;FOLD LIN P413 Vel=2 m/s CPDAT413 Tool[1]:marker Base[0] ;%{PE}
;FOLD Parameters ;%{h}
;Params IlfProvider=kukaroboter.basistech.inlineforms.movement.old; Kuka.IsGlobalPoint=False; Kuka.PointName=P413; Kuka.BlendingEnabled=False; Kuka.MoveDataName=CPDAT1; Kuka.VelocityPath=2; Kuka.CurrentCDSetIndex=0; Kuka.MovementParameterFieldEnabled=True; IlfCommand=LIN
;ENDFOLD
$BWDSTART = FALSE
LDAT_ACT = LCPDAT413
FDAT_ACT = FP413
BAS(#CP_PARAMS, 2.0)
SET_CD_PARAMS (0)
LIN XP413
;ENDFOLD

;FOLD LIN P414 Vel=2 m/s CPDAT414 Tool[1]:marker Base[0] ;%{PE}
;FOLD Parameters ;%{h}
;Params IlfProvider=kukaroboter.basistech.inlineforms.movement.old; Kuka.IsGlobalPoint=False; Kuka.PointName=P414; Kuka.BlendingEnabled=False; Kuka.MoveDataName=CPDAT1; Kuka.VelocityPath=2; Kuka.CurrentCDSetIndex=0; Kuka.MovementParameterFieldEnabled=True; IlfCommand=LIN
;ENDFOLD
$BWDSTART = FALSE
LDAT_ACT = LCPDAT414
FDAT_ACT = FP414
BAS(#CP_PARAMS, 2.0)
SET_CD_PARAMS (0)
LIN XP414
;ENDFOLD

;FOLD LIN P415 Vel=2 m/s CPDAT415 Tool[1]:marker Base[0] ;%{PE}
;FOLD Parameters ;%{h}
;Params IlfProvider=kukaroboter.basistech.inlineforms.movement.old; Kuka.IsGlobalPoint=False; Kuka.PointName=P415; Kuka.BlendingEnabled=False; Kuka.MoveDataName=CPDAT1; Kuka.VelocityPath=2; Kuka.CurrentCDSetIndex=0; Kuka.MovementParameterFieldEnabled=True; IlfCommand=LIN
;ENDFOLD
$BWDSTART = FALSE
LDAT_ACT = LCPDAT415
FDAT_ACT = FP415
BAS(#CP_PARAMS, 2.0)
SET_CD_PARAMS (0)
LIN XP415
;ENDFOLD

;FOLD LIN P416 Vel=2 m/s CPDAT416 Tool[1]:marker Base[0] ;%{PE}
;FOLD Parameters ;%{h}
;Params IlfProvider=kukaroboter.basistech.inlineforms.movement.old; Kuka.IsGlobalPoint=False; Kuka.PointName=P416; Kuka.BlendingEnabled=False; Kuka.MoveDataName=CPDAT1; Kuka.VelocityPath=2; Kuka.CurrentCDSetIndex=0; Kuka.MovementParameterFieldEnabled=True; IlfCommand=LIN
;ENDFOLD
$BWDSTART = FALSE
LDAT_ACT = LCPDAT416
FDAT_ACT = FP416
BAS(#CP_PARAMS, 2.0)
SET_CD_PARAMS (0)
LIN XP416
;ENDFOLD

;FOLD LIN P417 Vel=2 m/s CPDAT417 Tool[1]:marker Base[0] ;%{PE}
;FOLD Parameters ;%{h}
;Params IlfProvider=kukaroboter.basistech.inlineforms.movement.old; Kuka.IsGlobalPoint=False; Kuka.PointName=P417; Kuka.BlendingEnabled=False; Kuka.MoveDataName=CPDAT1; Kuka.VelocityPath=2; Kuka.CurrentCDSetIndex=0; Kuka.MovementParameterFieldEnabled=True; IlfCommand=LIN
;ENDFOLD
$BWDSTART = FALSE
LDAT_ACT = LCPDAT417
FDAT_ACT = FP417
BAS(#CP_PARAMS, 2.0)
SET_CD_PARAMS (0)
LIN XP417
;ENDFOLD

;FOLD LIN P418 Vel=2 m/s CPDAT418 Tool[1]:marker Base[0] ;%{PE}
;FOLD Parameters ;%{h}
;Params IlfProvider=kukaroboter.basistech.inlineforms.movement.old; Kuka.IsGlobalPoint=False; Kuka.PointName=P418; Kuka.BlendingEnabled=False; Kuka.MoveDataName=CPDAT1; Kuka.VelocityPath=2; Kuka.CurrentCDSetIndex=0; Kuka.MovementParameterFieldEnabled=True; IlfCommand=LIN
;ENDFOLD
$BWDSTART = FALSE
LDAT_ACT = LCPDAT418
FDAT_ACT = FP418
BAS(#CP_PARAMS, 2.0)
SET_CD_PARAMS (0)
LIN XP418
;ENDFOLD

;FOLD LIN P419 Vel=2 m/s CPDAT419 Tool[1]:marker Base[0] ;%{PE}
;FOLD Parameters ;%{h}
;Params IlfProvider=kukaroboter.basistech.inlineforms.movement.old; Kuka.IsGlobalPoint=False; Kuka.PointName=P419; Kuka.BlendingEnabled=False; Kuka.MoveDataName=CPDAT1; Kuka.VelocityPath=2; Kuka.CurrentCDSetIndex=0; Kuka.MovementParameterFieldEnabled=True; IlfCommand=LIN
;ENDFOLD
$BWDSTART = FALSE
LDAT_ACT = LCPDAT419
FDAT_ACT = FP419
BAS(#CP_PARAMS, 2.0)
SET_CD_PARAMS (0)
LIN XP419
;ENDFOLD

;FOLD LIN P420 Vel=2 m/s CPDAT420 Tool[1]:marker Base[0] ;%{PE}
;FOLD Parameters ;%{h}
;Params IlfProvider=kukaroboter.basistech.inlineforms.movement.old; Kuka.IsGlobalPoint=False; Kuka.PointName=P420; Kuka.BlendingEnabled=False; Kuka.MoveDataName=CPDAT1; Kuka.VelocityPath=2; Kuka.CurrentCDSetIndex=0; Kuka.MovementParameterFieldEnabled=True; IlfCommand=LIN
;ENDFOLD
$BWDSTART = FALSE
LDAT_ACT = LCPDAT420
FDAT_ACT = FP420
BAS(#CP_PARAMS, 2.0)
SET_CD_PARAMS (0)
LIN XP420
;ENDFOLD

;FOLD LIN P421 Vel=2 m/s CPDAT421 Tool[1]:marker Base[0] ;%{PE}
;FOLD Parameters ;%{h}
;Params IlfProvider=kukaroboter.basistech.inlineforms.movement.old; Kuka.IsGlobalPoint=False; Kuka.PointName=P421; Kuka.BlendingEnabled=False; Kuka.MoveDataName=CPDAT1; Kuka.VelocityPath=2; Kuka.CurrentCDSetIndex=0; Kuka.MovementParameterFieldEnabled=True; IlfCommand=LIN
;ENDFOLD
$BWDSTART = FALSE
LDAT_ACT = LCPDAT421
FDAT_ACT = FP421
BAS(#CP_PARAMS, 2.0)
SET_CD_PARAMS (0)
LIN XP421
;ENDFOLD

;FOLD LIN P422 Vel=2 m/s CPDAT422 Tool[1]:marker Base[0] ;%{PE}
;FOLD Parameters ;%{h}
;Params IlfProvider=kukaroboter.basistech.inlineforms.movement.old; Kuka.IsGlobalPoint=False; Kuka.PointName=P422; Kuka.BlendingEnabled=False; Kuka.MoveDataName=CPDAT1; Kuka.VelocityPath=2; Kuka.CurrentCDSetIndex=0; Kuka.MovementParameterFieldEnabled=True; IlfCommand=LIN
;ENDFOLD
$BWDSTART = FALSE
LDAT_ACT = LCPDAT422
FDAT_ACT = FP422
BAS(#CP_PARAMS, 2.0)
SET_CD_PARAMS (0)
LIN XP422
;ENDFOLD

;FOLD LIN P423 Vel=2 m/s CPDAT423 Tool[1]:marker Base[0] ;%{PE}
;FOLD Parameters ;%{h}
;Params IlfProvider=kukaroboter.basistech.inlineforms.movement.old; Kuka.IsGlobalPoint=False; Kuka.PointName=P423; Kuka.BlendingEnabled=False; Kuka.MoveDataName=CPDAT1; Kuka.VelocityPath=2; Kuka.CurrentCDSetIndex=0; Kuka.MovementParameterFieldEnabled=True; IlfCommand=LIN
;ENDFOLD
$BWDSTART = FALSE
LDAT_ACT = LCPDAT423
FDAT_ACT = FP423
BAS(#CP_PARAMS, 2.0)
SET_CD_PARAMS (0)
LIN XP423
;ENDFOLD

;FOLD LIN P424 Vel=2 m/s CPDAT424 Tool[1]:marker Base[0] ;%{PE}
;FOLD Parameters ;%{h}
;Params IlfProvider=kukaroboter.basistech.inlineforms.movement.old; Kuka.IsGlobalPoint=False; Kuka.PointName=P424; Kuka.BlendingEnabled=False; Kuka.MoveDataName=CPDAT1; Kuka.VelocityPath=2; Kuka.CurrentCDSetIndex=0; Kuka.MovementParameterFieldEnabled=True; IlfCommand=LIN
;ENDFOLD
$BWDSTART = FALSE
LDAT_ACT = LCPDAT424
FDAT_ACT = FP424
BAS(#CP_PARAMS, 2.0)
SET_CD_PARAMS (0)
LIN XP424
;ENDFOLD

;FOLD LIN P425 Vel=2 m/s CPDAT425 Tool[1]:marker Base[0] ;%{PE}
;FOLD Parameters ;%{h}
;Params IlfProvider=kukaroboter.basistech.inlineforms.movement.old; Kuka.IsGlobalPoint=False; Kuka.PointName=P425; Kuka.BlendingEnabled=False; Kuka.MoveDataName=CPDAT1; Kuka.VelocityPath=2; Kuka.CurrentCDSetIndex=0; Kuka.MovementParameterFieldEnabled=True; IlfCommand=LIN
;ENDFOLD
$BWDSTART = FALSE
LDAT_ACT = LCPDAT425
FDAT_ACT = FP425
BAS(#CP_PARAMS, 2.0)
SET_CD_PARAMS (0)
LIN XP425
;ENDFOLD

;FOLD LIN P426 Vel=2 m/s CPDAT426 Tool[1]:marker Base[0] ;%{PE}
;FOLD Parameters ;%{h}
;Params IlfProvider=kukaroboter.basistech.inlineforms.movement.old; Kuka.IsGlobalPoint=False; Kuka.PointName=P426; Kuka.BlendingEnabled=False; Kuka.MoveDataName=CPDAT1; Kuka.VelocityPath=2; Kuka.CurrentCDSetIndex=0; Kuka.MovementParameterFieldEnabled=True; IlfCommand=LIN
;ENDFOLD
$BWDSTART = FALSE
LDAT_ACT = LCPDAT426
FDAT_ACT = FP426
BAS(#CP_PARAMS, 2.0)
SET_CD_PARAMS (0)
LIN XP426
;ENDFOLD

;FOLD LIN P427 Vel=2 m/s CPDAT427 Tool[1]:marker Base[0] ;%{PE}
;FOLD Parameters ;%{h}
;Params IlfProvider=kukaroboter.basistech.inlineforms.movement.old; Kuka.IsGlobalPoint=False; Kuka.PointName=P427; Kuka.BlendingEnabled=False; Kuka.MoveDataName=CPDAT1; Kuka.VelocityPath=2; Kuka.CurrentCDSetIndex=0; Kuka.MovementParameterFieldEnabled=True; IlfCommand=LIN
;ENDFOLD
$BWDSTART = FALSE
LDAT_ACT = LCPDAT427
FDAT_ACT = FP427
BAS(#CP_PARAMS, 2.0)
SET_CD_PARAMS (0)
LIN XP427
;ENDFOLD

;FOLD LIN P428 Vel=2 m/s CPDAT428 Tool[1]:marker Base[0] ;%{PE}
;FOLD Parameters ;%{h}
;Params IlfProvider=kukaroboter.basistech.inlineforms.movement.old; Kuka.IsGlobalPoint=False; Kuka.PointName=P428; Kuka.BlendingEnabled=False; Kuka.MoveDataName=CPDAT1; Kuka.VelocityPath=2; Kuka.CurrentCDSetIndex=0; Kuka.MovementParameterFieldEnabled=True; IlfCommand=LIN
;ENDFOLD
$BWDSTART = FALSE
LDAT_ACT = LCPDAT428
FDAT_ACT = FP428
BAS(#CP_PARAMS, 2.0)
SET_CD_PARAMS (0)
LIN XP428
;ENDFOLD

;FOLD LIN P429 Vel=2 m/s CPDAT429 Tool[1]:marker Base[0] ;%{PE}
;FOLD Parameters ;%{h}
;Params IlfProvider=kukaroboter.basistech.inlineforms.movement.old; Kuka.IsGlobalPoint=False; Kuka.PointName=P429; Kuka.BlendingEnabled=False; Kuka.MoveDataName=CPDAT1; Kuka.VelocityPath=2; Kuka.CurrentCDSetIndex=0; Kuka.MovementParameterFieldEnabled=True; IlfCommand=LIN
;ENDFOLD
$BWDSTART = FALSE
LDAT_ACT = LCPDAT429
FDAT_ACT = FP429
BAS(#CP_PARAMS, 2.0)
SET_CD_PARAMS (0)
LIN XP429
;ENDFOLD

;FOLD LIN P430 Vel=2 m/s CPDAT430 Tool[1]:marker Base[0] ;%{PE}
;FOLD Parameters ;%{h}
;Params IlfProvider=kukaroboter.basistech.inlineforms.movement.old; Kuka.IsGlobalPoint=False; Kuka.PointName=P430; Kuka.BlendingEnabled=False; Kuka.MoveDataName=CPDAT1; Kuka.VelocityPath=2; Kuka.CurrentCDSetIndex=0; Kuka.MovementParameterFieldEnabled=True; IlfCommand=LIN
;ENDFOLD
$BWDSTART = FALSE
LDAT_ACT = LCPDAT430
FDAT_ACT = FP430
BAS(#CP_PARAMS, 2.0)
SET_CD_PARAMS (0)
LIN XP430
;ENDFOLD

;FOLD LIN P431 Vel=2 m/s CPDAT431 Tool[1]:marker Base[0] ;%{PE}
;FOLD Parameters ;%{h}
;Params IlfProvider=kukaroboter.basistech.inlineforms.movement.old; Kuka.IsGlobalPoint=False; Kuka.PointName=P431; Kuka.BlendingEnabled=False; Kuka.MoveDataName=CPDAT1; Kuka.VelocityPath=2; Kuka.CurrentCDSetIndex=0; Kuka.MovementParameterFieldEnabled=True; IlfCommand=LIN
;ENDFOLD
$BWDSTART = FALSE
LDAT_ACT = LCPDAT431
FDAT_ACT = FP431
BAS(#CP_PARAMS, 2.0)
SET_CD_PARAMS (0)
LIN XP431
;ENDFOLD

;FOLD LIN P432 Vel=2 m/s CPDAT432 Tool[1]:marker Base[0] ;%{PE}
;FOLD Parameters ;%{h}
;Params IlfProvider=kukaroboter.basistech.inlineforms.movement.old; Kuka.IsGlobalPoint=False; Kuka.PointName=P432; Kuka.BlendingEnabled=False; Kuka.MoveDataName=CPDAT1; Kuka.VelocityPath=2; Kuka.CurrentCDSetIndex=0; Kuka.MovementParameterFieldEnabled=True; IlfCommand=LIN
;ENDFOLD
$BWDSTART = FALSE
LDAT_ACT = LCPDAT432
FDAT_ACT = FP432
BAS(#CP_PARAMS, 2.0)
SET_CD_PARAMS (0)
LIN XP432
;ENDFOLD

;FOLD LIN P433 Vel=2 m/s CPDAT433 Tool[1]:marker Base[0] ;%{PE}
;FOLD Parameters ;%{h}
;Params IlfProvider=kukaroboter.basistech.inlineforms.movement.old; Kuka.IsGlobalPoint=False; Kuka.PointName=P433; Kuka.BlendingEnabled=False; Kuka.MoveDataName=CPDAT1; Kuka.VelocityPath=2; Kuka.CurrentCDSetIndex=0; Kuka.MovementParameterFieldEnabled=True; IlfCommand=LIN
;ENDFOLD
$BWDSTART = FALSE
LDAT_ACT = LCPDAT433
FDAT_ACT = FP433
BAS(#CP_PARAMS, 2.0)
SET_CD_PARAMS (0)
LIN XP433
;ENDFOLD

;FOLD LIN P434 Vel=2 m/s CPDAT434 Tool[1]:marker Base[0] ;%{PE}
;FOLD Parameters ;%{h}
;Params IlfProvider=kukaroboter.basistech.inlineforms.movement.old; Kuka.IsGlobalPoint=False; Kuka.PointName=P434; Kuka.BlendingEnabled=False; Kuka.MoveDataName=CPDAT1; Kuka.VelocityPath=2; Kuka.CurrentCDSetIndex=0; Kuka.MovementParameterFieldEnabled=True; IlfCommand=LIN
;ENDFOLD
$BWDSTART = FALSE
LDAT_ACT = LCPDAT434
FDAT_ACT = FP434
BAS(#CP_PARAMS, 2.0)
SET_CD_PARAMS (0)
LIN XP434
;ENDFOLD

;FOLD LIN P435 Vel=2 m/s CPDAT435 Tool[1]:marker Base[0] ;%{PE}
;FOLD Parameters ;%{h}
;Params IlfProvider=kukaroboter.basistech.inlineforms.movement.old; Kuka.IsGlobalPoint=False; Kuka.PointName=P435; Kuka.BlendingEnabled=False; Kuka.MoveDataName=CPDAT1; Kuka.VelocityPath=2; Kuka.CurrentCDSetIndex=0; Kuka.MovementParameterFieldEnabled=True; IlfCommand=LIN
;ENDFOLD
$BWDSTART = FALSE
LDAT_ACT = LCPDAT435
FDAT_ACT = FP435
BAS(#CP_PARAMS, 2.0)
SET_CD_PARAMS (0)
LIN XP435
;ENDFOLD

;FOLD LIN P436 Vel=2 m/s CPDAT436 Tool[1]:marker Base[0] ;%{PE}
;FOLD Parameters ;%{h}
;Params IlfProvider=kukaroboter.basistech.inlineforms.movement.old; Kuka.IsGlobalPoint=False; Kuka.PointName=P436; Kuka.BlendingEnabled=False; Kuka.MoveDataName=CPDAT1; Kuka.VelocityPath=2; Kuka.CurrentCDSetIndex=0; Kuka.MovementParameterFieldEnabled=True; IlfCommand=LIN
;ENDFOLD
$BWDSTART = FALSE
LDAT_ACT = LCPDAT436
FDAT_ACT = FP436
BAS(#CP_PARAMS, 2.0)
SET_CD_PARAMS (0)
LIN XP436
;ENDFOLD

;FOLD LIN P437 Vel=2 m/s CPDAT437 Tool[1]:marker Base[0] ;%{PE}
;FOLD Parameters ;%{h}
;Params IlfProvider=kukaroboter.basistech.inlineforms.movement.old; Kuka.IsGlobalPoint=False; Kuka.PointName=P437; Kuka.BlendingEnabled=False; Kuka.MoveDataName=CPDAT1; Kuka.VelocityPath=2; Kuka.CurrentCDSetIndex=0; Kuka.MovementParameterFieldEnabled=True; IlfCommand=LIN
;ENDFOLD
$BWDSTART = FALSE
LDAT_ACT = LCPDAT437
FDAT_ACT = FP437
BAS(#CP_PARAMS, 2.0)
SET_CD_PARAMS (0)
LIN XP437
;ENDFOLD

;FOLD LIN P438 Vel=2 m/s CPDAT438 Tool[1]:marker Base[0] ;%{PE}
;FOLD Parameters ;%{h}
;Params IlfProvider=kukaroboter.basistech.inlineforms.movement.old; Kuka.IsGlobalPoint=False; Kuka.PointName=P438; Kuka.BlendingEnabled=False; Kuka.MoveDataName=CPDAT1; Kuka.VelocityPath=2; Kuka.CurrentCDSetIndex=0; Kuka.MovementParameterFieldEnabled=True; IlfCommand=LIN
;ENDFOLD
$BWDSTART = FALSE
LDAT_ACT = LCPDAT438
FDAT_ACT = FP438
BAS(#CP_PARAMS, 2.0)
SET_CD_PARAMS (0)
LIN XP438
;ENDFOLD

;FOLD LIN P439 Vel=2 m/s CPDAT439 Tool[1]:marker Base[0] ;%{PE}
;FOLD Parameters ;%{h}
;Params IlfProvider=kukaroboter.basistech.inlineforms.movement.old; Kuka.IsGlobalPoint=False; Kuka.PointName=P439; Kuka.BlendingEnabled=False; Kuka.MoveDataName=CPDAT1; Kuka.VelocityPath=2; Kuka.CurrentCDSetIndex=0; Kuka.MovementParameterFieldEnabled=True; IlfCommand=LIN
;ENDFOLD
$BWDSTART = FALSE
LDAT_ACT = LCPDAT439
FDAT_ACT = FP439
BAS(#CP_PARAMS, 2.0)
SET_CD_PARAMS (0)
LIN XP439
;ENDFOLD

;FOLD LIN P440 Vel=2 m/s CPDAT440 Tool[1]:marker Base[0] ;%{PE}
;FOLD Parameters ;%{h}
;Params IlfProvider=kukaroboter.basistech.inlineforms.movement.old; Kuka.IsGlobalPoint=False; Kuka.PointName=P440; Kuka.BlendingEnabled=False; Kuka.MoveDataName=CPDAT1; Kuka.VelocityPath=2; Kuka.CurrentCDSetIndex=0; Kuka.MovementParameterFieldEnabled=True; IlfCommand=LIN
;ENDFOLD
$BWDSTART = FALSE
LDAT_ACT = LCPDAT440
FDAT_ACT = FP440
BAS(#CP_PARAMS, 2.0)
SET_CD_PARAMS (0)
LIN XP440
;ENDFOLD

;FOLD LIN P441 Vel=2 m/s CPDAT441 Tool[1]:marker Base[0] ;%{PE}
;FOLD Parameters ;%{h}
;Params IlfProvider=kukaroboter.basistech.inlineforms.movement.old; Kuka.IsGlobalPoint=False; Kuka.PointName=P441; Kuka.BlendingEnabled=False; Kuka.MoveDataName=CPDAT1; Kuka.VelocityPath=2; Kuka.CurrentCDSetIndex=0; Kuka.MovementParameterFieldEnabled=True; IlfCommand=LIN
;ENDFOLD
$BWDSTART = FALSE
LDAT_ACT = LCPDAT441
FDAT_ACT = FP441
BAS(#CP_PARAMS, 2.0)
SET_CD_PARAMS (0)
LIN XP441
;ENDFOLD

;FOLD LIN P442 Vel=2 m/s CPDAT442 Tool[1]:marker Base[0] ;%{PE}
;FOLD Parameters ;%{h}
;Params IlfProvider=kukaroboter.basistech.inlineforms.movement.old; Kuka.IsGlobalPoint=False; Kuka.PointName=P442; Kuka.BlendingEnabled=False; Kuka.MoveDataName=CPDAT1; Kuka.VelocityPath=2; Kuka.CurrentCDSetIndex=0; Kuka.MovementParameterFieldEnabled=True; IlfCommand=LIN
;ENDFOLD
$BWDSTART = FALSE
LDAT_ACT = LCPDAT442
FDAT_ACT = FP442
BAS(#CP_PARAMS, 2.0)
SET_CD_PARAMS (0)
LIN XP442
;ENDFOLD

;FOLD LIN P443 Vel=2 m/s CPDAT443 Tool[1]:marker Base[0] ;%{PE}
;FOLD Parameters ;%{h}
;Params IlfProvider=kukaroboter.basistech.inlineforms.movement.old; Kuka.IsGlobalPoint=False; Kuka.PointName=P443; Kuka.BlendingEnabled=False; Kuka.MoveDataName=CPDAT1; Kuka.VelocityPath=2; Kuka.CurrentCDSetIndex=0; Kuka.MovementParameterFieldEnabled=True; IlfCommand=LIN
;ENDFOLD
$BWDSTART = FALSE
LDAT_ACT = LCPDAT443
FDAT_ACT = FP443
BAS(#CP_PARAMS, 2.0)
SET_CD_PARAMS (0)
LIN XP443
;ENDFOLD

;FOLD LIN P444 Vel=2 m/s CPDAT444 Tool[1]:marker Base[0] ;%{PE}
;FOLD Parameters ;%{h}
;Params IlfProvider=kukaroboter.basistech.inlineforms.movement.old; Kuka.IsGlobalPoint=False; Kuka.PointName=P444; Kuka.BlendingEnabled=False; Kuka.MoveDataName=CPDAT1; Kuka.VelocityPath=2; Kuka.CurrentCDSetIndex=0; Kuka.MovementParameterFieldEnabled=True; IlfCommand=LIN
;ENDFOLD
$BWDSTART = FALSE
LDAT_ACT = LCPDAT444
FDAT_ACT = FP444
BAS(#CP_PARAMS, 2.0)
SET_CD_PARAMS (0)
LIN XP444
;ENDFOLD

;FOLD LIN P445 Vel=2 m/s CPDAT445 Tool[1]:marker Base[0] ;%{PE}
;FOLD Parameters ;%{h}
;Params IlfProvider=kukaroboter.basistech.inlineforms.movement.old; Kuka.IsGlobalPoint=False; Kuka.PointName=P445; Kuka.BlendingEnabled=False; Kuka.MoveDataName=CPDAT1; Kuka.VelocityPath=2; Kuka.CurrentCDSetIndex=0; Kuka.MovementParameterFieldEnabled=True; IlfCommand=LIN
;ENDFOLD
$BWDSTART = FALSE
LDAT_ACT = LCPDAT445
FDAT_ACT = FP445
BAS(#CP_PARAMS, 2.0)
SET_CD_PARAMS (0)
LIN XP445
;ENDFOLD

;FOLD LIN P446 Vel=2 m/s CPDAT446 Tool[1]:marker Base[0] ;%{PE}
;FOLD Parameters ;%{h}
;Params IlfProvider=kukaroboter.basistech.inlineforms.movement.old; Kuka.IsGlobalPoint=False; Kuka.PointName=P446; Kuka.BlendingEnabled=False; Kuka.MoveDataName=CPDAT1; Kuka.VelocityPath=2; Kuka.CurrentCDSetIndex=0; Kuka.MovementParameterFieldEnabled=True; IlfCommand=LIN
;ENDFOLD
$BWDSTART = FALSE
LDAT_ACT = LCPDAT446
FDAT_ACT = FP446
BAS(#CP_PARAMS, 2.0)
SET_CD_PARAMS (0)
LIN XP446
;ENDFOLD

;FOLD LIN P447 Vel=2 m/s CPDAT447 Tool[1]:marker Base[0] ;%{PE}
;FOLD Parameters ;%{h}
;Params IlfProvider=kukaroboter.basistech.inlineforms.movement.old; Kuka.IsGlobalPoint=False; Kuka.PointName=P447; Kuka.BlendingEnabled=False; Kuka.MoveDataName=CPDAT1; Kuka.VelocityPath=2; Kuka.CurrentCDSetIndex=0; Kuka.MovementParameterFieldEnabled=True; IlfCommand=LIN
;ENDFOLD
$BWDSTART = FALSE
LDAT_ACT = LCPDAT447
FDAT_ACT = FP447
BAS(#CP_PARAMS, 2.0)
SET_CD_PARAMS (0)
LIN XP447
;ENDFOLD

;FOLD LIN P448 Vel=2 m/s CPDAT448 Tool[1]:marker Base[0] ;%{PE}
;FOLD Parameters ;%{h}
;Params IlfProvider=kukaroboter.basistech.inlineforms.movement.old; Kuka.IsGlobalPoint=False; Kuka.PointName=P448; Kuka.BlendingEnabled=False; Kuka.MoveDataName=CPDAT1; Kuka.VelocityPath=2; Kuka.CurrentCDSetIndex=0; Kuka.MovementParameterFieldEnabled=True; IlfCommand=LIN
;ENDFOLD
$BWDSTART = FALSE
LDAT_ACT = LCPDAT448
FDAT_ACT = FP448
BAS(#CP_PARAMS, 2.0)
SET_CD_PARAMS (0)
LIN XP448
;ENDFOLD

;FOLD LIN P449 Vel=2 m/s CPDAT449 Tool[1]:marker Base[0] ;%{PE}
;FOLD Parameters ;%{h}
;Params IlfProvider=kukaroboter.basistech.inlineforms.movement.old; Kuka.IsGlobalPoint=False; Kuka.PointName=P449; Kuka.BlendingEnabled=False; Kuka.MoveDataName=CPDAT1; Kuka.VelocityPath=2; Kuka.CurrentCDSetIndex=0; Kuka.MovementParameterFieldEnabled=True; IlfCommand=LIN
;ENDFOLD
$BWDSTART = FALSE
LDAT_ACT = LCPDAT449
FDAT_ACT = FP449
BAS(#CP_PARAMS, 2.0)
SET_CD_PARAMS (0)
LIN XP449
;ENDFOLD

;FOLD LIN P450 Vel=2 m/s CPDAT450 Tool[1]:marker Base[0] ;%{PE}
;FOLD Parameters ;%{h}
;Params IlfProvider=kukaroboter.basistech.inlineforms.movement.old; Kuka.IsGlobalPoint=False; Kuka.PointName=P450; Kuka.BlendingEnabled=False; Kuka.MoveDataName=CPDAT1; Kuka.VelocityPath=2; Kuka.CurrentCDSetIndex=0; Kuka.MovementParameterFieldEnabled=True; IlfCommand=LIN
;ENDFOLD
$BWDSTART = FALSE
LDAT_ACT = LCPDAT450
FDAT_ACT = FP450
BAS(#CP_PARAMS, 2.0)
SET_CD_PARAMS (0)
LIN XP450
;ENDFOLD

;FOLD LIN P451 Vel=2 m/s CPDAT451 Tool[1]:marker Base[0] ;%{PE}
;FOLD Parameters ;%{h}
;Params IlfProvider=kukaroboter.basistech.inlineforms.movement.old; Kuka.IsGlobalPoint=False; Kuka.PointName=P451; Kuka.BlendingEnabled=False; Kuka.MoveDataName=CPDAT1; Kuka.VelocityPath=2; Kuka.CurrentCDSetIndex=0; Kuka.MovementParameterFieldEnabled=True; IlfCommand=LIN
;ENDFOLD
$BWDSTART = FALSE
LDAT_ACT = LCPDAT451
FDAT_ACT = FP451
BAS(#CP_PARAMS, 2.0)
SET_CD_PARAMS (0)
LIN XP451
;ENDFOLD

;FOLD LIN P452 Vel=2 m/s CPDAT452 Tool[1]:marker Base[0] ;%{PE}
;FOLD Parameters ;%{h}
;Params IlfProvider=kukaroboter.basistech.inlineforms.movement.old; Kuka.IsGlobalPoint=False; Kuka.PointName=P452; Kuka.BlendingEnabled=False; Kuka.MoveDataName=CPDAT1; Kuka.VelocityPath=2; Kuka.CurrentCDSetIndex=0; Kuka.MovementParameterFieldEnabled=True; IlfCommand=LIN
;ENDFOLD
$BWDSTART = FALSE
LDAT_ACT = LCPDAT452
FDAT_ACT = FP452
BAS(#CP_PARAMS, 2.0)
SET_CD_PARAMS (0)
LIN XP452
;ENDFOLD

;FOLD LIN P453 Vel=2 m/s CPDAT453 Tool[1]:marker Base[0] ;%{PE}
;FOLD Parameters ;%{h}
;Params IlfProvider=kukaroboter.basistech.inlineforms.movement.old; Kuka.IsGlobalPoint=False; Kuka.PointName=P453; Kuka.BlendingEnabled=False; Kuka.MoveDataName=CPDAT1; Kuka.VelocityPath=2; Kuka.CurrentCDSetIndex=0; Kuka.MovementParameterFieldEnabled=True; IlfCommand=LIN
;ENDFOLD
$BWDSTART = FALSE
LDAT_ACT = LCPDAT453
FDAT_ACT = FP453
BAS(#CP_PARAMS, 2.0)
SET_CD_PARAMS (0)
LIN XP453
;ENDFOLD

;FOLD LIN P454 Vel=2 m/s CPDAT454 Tool[1]:marker Base[0] ;%{PE}
;FOLD Parameters ;%{h}
;Params IlfProvider=kukaroboter.basistech.inlineforms.movement.old; Kuka.IsGlobalPoint=False; Kuka.PointName=P454; Kuka.BlendingEnabled=False; Kuka.MoveDataName=CPDAT1; Kuka.VelocityPath=2; Kuka.CurrentCDSetIndex=0; Kuka.MovementParameterFieldEnabled=True; IlfCommand=LIN
;ENDFOLD
$BWDSTART = FALSE
LDAT_ACT = LCPDAT454
FDAT_ACT = FP454
BAS(#CP_PARAMS, 2.0)
SET_CD_PARAMS (0)
LIN XP454
;ENDFOLD

;FOLD LIN P455 Vel=2 m/s CPDAT455 Tool[1]:marker Base[0] ;%{PE}
;FOLD Parameters ;%{h}
;Params IlfProvider=kukaroboter.basistech.inlineforms.movement.old; Kuka.IsGlobalPoint=False; Kuka.PointName=P455; Kuka.BlendingEnabled=False; Kuka.MoveDataName=CPDAT1; Kuka.VelocityPath=2; Kuka.CurrentCDSetIndex=0; Kuka.MovementParameterFieldEnabled=True; IlfCommand=LIN
;ENDFOLD
$BWDSTART = FALSE
LDAT_ACT = LCPDAT455
FDAT_ACT = FP455
BAS(#CP_PARAMS, 2.0)
SET_CD_PARAMS (0)
LIN XP455
;ENDFOLD

;FOLD LIN P456 Vel=2 m/s CPDAT456 Tool[1]:marker Base[0] ;%{PE}
;FOLD Parameters ;%{h}
;Params IlfProvider=kukaroboter.basistech.inlineforms.movement.old; Kuka.IsGlobalPoint=False; Kuka.PointName=P456; Kuka.BlendingEnabled=False; Kuka.MoveDataName=CPDAT1; Kuka.VelocityPath=2; Kuka.CurrentCDSetIndex=0; Kuka.MovementParameterFieldEnabled=True; IlfCommand=LIN
;ENDFOLD
$BWDSTART = FALSE
LDAT_ACT = LCPDAT456
FDAT_ACT = FP456
BAS(#CP_PARAMS, 2.0)
SET_CD_PARAMS (0)
LIN XP456
;ENDFOLD

;FOLD LIN P457 Vel=2 m/s CPDAT457 Tool[1]:marker Base[0] ;%{PE}
;FOLD Parameters ;%{h}
;Params IlfProvider=kukaroboter.basistech.inlineforms.movement.old; Kuka.IsGlobalPoint=False; Kuka.PointName=P457; Kuka.BlendingEnabled=False; Kuka.MoveDataName=CPDAT1; Kuka.VelocityPath=2; Kuka.CurrentCDSetIndex=0; Kuka.MovementParameterFieldEnabled=True; IlfCommand=LIN
;ENDFOLD
$BWDSTART = FALSE
LDAT_ACT = LCPDAT457
FDAT_ACT = FP457
BAS(#CP_PARAMS, 2.0)
SET_CD_PARAMS (0)
LIN XP457
;ENDFOLD

;FOLD LIN P458 Vel=2 m/s CPDAT458 Tool[1]:marker Base[0] ;%{PE}
;FOLD Parameters ;%{h}
;Params IlfProvider=kukaroboter.basistech.inlineforms.movement.old; Kuka.IsGlobalPoint=False; Kuka.PointName=P458; Kuka.BlendingEnabled=False; Kuka.MoveDataName=CPDAT1; Kuka.VelocityPath=2; Kuka.CurrentCDSetIndex=0; Kuka.MovementParameterFieldEnabled=True; IlfCommand=LIN
;ENDFOLD
$BWDSTART = FALSE
LDAT_ACT = LCPDAT458
FDAT_ACT = FP458
BAS(#CP_PARAMS, 2.0)
SET_CD_PARAMS (0)
LIN XP458
;ENDFOLD

;FOLD LIN P459 Vel=2 m/s CPDAT459 Tool[1]:marker Base[0] ;%{PE}
;FOLD Parameters ;%{h}
;Params IlfProvider=kukaroboter.basistech.inlineforms.movement.old; Kuka.IsGlobalPoint=False; Kuka.PointName=P459; Kuka.BlendingEnabled=False; Kuka.MoveDataName=CPDAT1; Kuka.VelocityPath=2; Kuka.CurrentCDSetIndex=0; Kuka.MovementParameterFieldEnabled=True; IlfCommand=LIN
;ENDFOLD
$BWDSTART = FALSE
LDAT_ACT = LCPDAT459
FDAT_ACT = FP459
BAS(#CP_PARAMS, 2.0)
SET_CD_PARAMS (0)
LIN XP459
;ENDFOLD

;FOLD LIN P460 Vel=2 m/s CPDAT460 Tool[1]:marker Base[0] ;%{PE}
;FOLD Parameters ;%{h}
;Params IlfProvider=kukaroboter.basistech.inlineforms.movement.old; Kuka.IsGlobalPoint=False; Kuka.PointName=P460; Kuka.BlendingEnabled=False; Kuka.MoveDataName=CPDAT1; Kuka.VelocityPath=2; Kuka.CurrentCDSetIndex=0; Kuka.MovementParameterFieldEnabled=True; IlfCommand=LIN
;ENDFOLD
$BWDSTART = FALSE
LDAT_ACT = LCPDAT460
FDAT_ACT = FP460
BAS(#CP_PARAMS, 2.0)
SET_CD_PARAMS (0)
LIN XP460
;ENDFOLD

;FOLD LIN P461 Vel=2 m/s CPDAT461 Tool[1]:marker Base[0] ;%{PE}
;FOLD Parameters ;%{h}
;Params IlfProvider=kukaroboter.basistech.inlineforms.movement.old; Kuka.IsGlobalPoint=False; Kuka.PointName=P461; Kuka.BlendingEnabled=False; Kuka.MoveDataName=CPDAT1; Kuka.VelocityPath=2; Kuka.CurrentCDSetIndex=0; Kuka.MovementParameterFieldEnabled=True; IlfCommand=LIN
;ENDFOLD
$BWDSTART = FALSE
LDAT_ACT = LCPDAT461
FDAT_ACT = FP461
BAS(#CP_PARAMS, 2.0)
SET_CD_PARAMS (0)
LIN XP461
;ENDFOLD

;FOLD LIN P462 Vel=2 m/s CPDAT462 Tool[1]:marker Base[0] ;%{PE}
;FOLD Parameters ;%{h}
;Params IlfProvider=kukaroboter.basistech.inlineforms.movement.old; Kuka.IsGlobalPoint=False; Kuka.PointName=P462; Kuka.BlendingEnabled=False; Kuka.MoveDataName=CPDAT1; Kuka.VelocityPath=2; Kuka.CurrentCDSetIndex=0; Kuka.MovementParameterFieldEnabled=True; IlfCommand=LIN
;ENDFOLD
$BWDSTART = FALSE
LDAT_ACT = LCPDAT462
FDAT_ACT = FP462
BAS(#CP_PARAMS, 2.0)
SET_CD_PARAMS (0)
LIN XP462
;ENDFOLD

;FOLD LIN P463 Vel=2 m/s CPDAT463 Tool[1]:marker Base[0] ;%{PE}
;FOLD Parameters ;%{h}
;Params IlfProvider=kukaroboter.basistech.inlineforms.movement.old; Kuka.IsGlobalPoint=False; Kuka.PointName=P463; Kuka.BlendingEnabled=False; Kuka.MoveDataName=CPDAT1; Kuka.VelocityPath=2; Kuka.CurrentCDSetIndex=0; Kuka.MovementParameterFieldEnabled=True; IlfCommand=LIN
;ENDFOLD
$BWDSTART = FALSE
LDAT_ACT = LCPDAT463
FDAT_ACT = FP463
BAS(#CP_PARAMS, 2.0)
SET_CD_PARAMS (0)
LIN XP463
;ENDFOLD

;FOLD LIN P464 Vel=2 m/s CPDAT464 Tool[1]:marker Base[0] ;%{PE}
;FOLD Parameters ;%{h}
;Params IlfProvider=kukaroboter.basistech.inlineforms.movement.old; Kuka.IsGlobalPoint=False; Kuka.PointName=P464; Kuka.BlendingEnabled=False; Kuka.MoveDataName=CPDAT1; Kuka.VelocityPath=2; Kuka.CurrentCDSetIndex=0; Kuka.MovementParameterFieldEnabled=True; IlfCommand=LIN
;ENDFOLD
$BWDSTART = FALSE
LDAT_ACT = LCPDAT464
FDAT_ACT = FP464
BAS(#CP_PARAMS, 2.0)
SET_CD_PARAMS (0)
LIN XP464
;ENDFOLD

;FOLD LIN P465 Vel=2 m/s CPDAT465 Tool[1]:marker Base[0] ;%{PE}
;FOLD Parameters ;%{h}
;Params IlfProvider=kukaroboter.basistech.inlineforms.movement.old; Kuka.IsGlobalPoint=False; Kuka.PointName=P465; Kuka.BlendingEnabled=False; Kuka.MoveDataName=CPDAT1; Kuka.VelocityPath=2; Kuka.CurrentCDSetIndex=0; Kuka.MovementParameterFieldEnabled=True; IlfCommand=LIN
;ENDFOLD
$BWDSTART = FALSE
LDAT_ACT = LCPDAT465
FDAT_ACT = FP465
BAS(#CP_PARAMS, 2.0)
SET_CD_PARAMS (0)
LIN XP465
;ENDFOLD

;FOLD LIN P466 Vel=2 m/s CPDAT466 Tool[1]:marker Base[0] ;%{PE}
;FOLD Parameters ;%{h}
;Params IlfProvider=kukaroboter.basistech.inlineforms.movement.old; Kuka.IsGlobalPoint=False; Kuka.PointName=P466; Kuka.BlendingEnabled=False; Kuka.MoveDataName=CPDAT1; Kuka.VelocityPath=2; Kuka.CurrentCDSetIndex=0; Kuka.MovementParameterFieldEnabled=True; IlfCommand=LIN
;ENDFOLD
$BWDSTART = FALSE
LDAT_ACT = LCPDAT466
FDAT_ACT = FP466
BAS(#CP_PARAMS, 2.0)
SET_CD_PARAMS (0)
LIN XP466
;ENDFOLD

;FOLD LIN P467 Vel=2 m/s CPDAT467 Tool[1]:marker Base[0] ;%{PE}
;FOLD Parameters ;%{h}
;Params IlfProvider=kukaroboter.basistech.inlineforms.movement.old; Kuka.IsGlobalPoint=False; Kuka.PointName=P467; Kuka.BlendingEnabled=False; Kuka.MoveDataName=CPDAT1; Kuka.VelocityPath=2; Kuka.CurrentCDSetIndex=0; Kuka.MovementParameterFieldEnabled=True; IlfCommand=LIN
;ENDFOLD
$BWDSTART = FALSE
LDAT_ACT = LCPDAT467
FDAT_ACT = FP467
BAS(#CP_PARAMS, 2.0)
SET_CD_PARAMS (0)
LIN XP467
;ENDFOLD

;FOLD LIN P468 Vel=2 m/s CPDAT468 Tool[1]:marker Base[0] ;%{PE}
;FOLD Parameters ;%{h}
;Params IlfProvider=kukaroboter.basistech.inlineforms.movement.old; Kuka.IsGlobalPoint=False; Kuka.PointName=P468; Kuka.BlendingEnabled=False; Kuka.MoveDataName=CPDAT1; Kuka.VelocityPath=2; Kuka.CurrentCDSetIndex=0; Kuka.MovementParameterFieldEnabled=True; IlfCommand=LIN
;ENDFOLD
$BWDSTART = FALSE
LDAT_ACT = LCPDAT468
FDAT_ACT = FP468
BAS(#CP_PARAMS, 2.0)
SET_CD_PARAMS (0)
LIN XP468
;ENDFOLD

;FOLD LIN P469 Vel=2 m/s CPDAT469 Tool[1]:marker Base[0] ;%{PE}
;FOLD Parameters ;%{h}
;Params IlfProvider=kukaroboter.basistech.inlineforms.movement.old; Kuka.IsGlobalPoint=False; Kuka.PointName=P469; Kuka.BlendingEnabled=False; Kuka.MoveDataName=CPDAT1; Kuka.VelocityPath=2; Kuka.CurrentCDSetIndex=0; Kuka.MovementParameterFieldEnabled=True; IlfCommand=LIN
;ENDFOLD
$BWDSTART = FALSE
LDAT_ACT = LCPDAT469
FDAT_ACT = FP469
BAS(#CP_PARAMS, 2.0)
SET_CD_PARAMS (0)
LIN XP469
;ENDFOLD

;FOLD LIN P470 Vel=2 m/s CPDAT470 Tool[1]:marker Base[0] ;%{PE}
;FOLD Parameters ;%{h}
;Params IlfProvider=kukaroboter.basistech.inlineforms.movement.old; Kuka.IsGlobalPoint=False; Kuka.PointName=P470; Kuka.BlendingEnabled=False; Kuka.MoveDataName=CPDAT1; Kuka.VelocityPath=2; Kuka.CurrentCDSetIndex=0; Kuka.MovementParameterFieldEnabled=True; IlfCommand=LIN
;ENDFOLD
$BWDSTART = FALSE
LDAT_ACT = LCPDAT470
FDAT_ACT = FP470
BAS(#CP_PARAMS, 2.0)
SET_CD_PARAMS (0)
LIN XP470
;ENDFOLD

;FOLD LIN P471 Vel=2 m/s CPDAT471 Tool[1]:marker Base[0] ;%{PE}
;FOLD Parameters ;%{h}
;Params IlfProvider=kukaroboter.basistech.inlineforms.movement.old; Kuka.IsGlobalPoint=False; Kuka.PointName=P471; Kuka.BlendingEnabled=False; Kuka.MoveDataName=CPDAT1; Kuka.VelocityPath=2; Kuka.CurrentCDSetIndex=0; Kuka.MovementParameterFieldEnabled=True; IlfCommand=LIN
;ENDFOLD
$BWDSTART = FALSE
LDAT_ACT = LCPDAT471
FDAT_ACT = FP471
BAS(#CP_PARAMS, 2.0)
SET_CD_PARAMS (0)
LIN XP471
;ENDFOLD

;FOLD LIN P472 Vel=2 m/s CPDAT472 Tool[1]:marker Base[0] ;%{PE}
;FOLD Parameters ;%{h}
;Params IlfProvider=kukaroboter.basistech.inlineforms.movement.old; Kuka.IsGlobalPoint=False; Kuka.PointName=P472; Kuka.BlendingEnabled=False; Kuka.MoveDataName=CPDAT1; Kuka.VelocityPath=2; Kuka.CurrentCDSetIndex=0; Kuka.MovementParameterFieldEnabled=True; IlfCommand=LIN
;ENDFOLD
$BWDSTART = FALSE
LDAT_ACT = LCPDAT472
FDAT_ACT = FP472
BAS(#CP_PARAMS, 2.0)
SET_CD_PARAMS (0)
LIN XP472
;ENDFOLD

;FOLD LIN P473 Vel=2 m/s CPDAT473 Tool[1]:marker Base[0] ;%{PE}
;FOLD Parameters ;%{h}
;Params IlfProvider=kukaroboter.basistech.inlineforms.movement.old; Kuka.IsGlobalPoint=False; Kuka.PointName=P473; Kuka.BlendingEnabled=False; Kuka.MoveDataName=CPDAT1; Kuka.VelocityPath=2; Kuka.CurrentCDSetIndex=0; Kuka.MovementParameterFieldEnabled=True; IlfCommand=LIN
;ENDFOLD
$BWDSTART = FALSE
LDAT_ACT = LCPDAT473
FDAT_ACT = FP473
BAS(#CP_PARAMS, 2.0)
SET_CD_PARAMS (0)
LIN XP473
;ENDFOLD

;FOLD LIN P474 Vel=2 m/s CPDAT474 Tool[1]:marker Base[0] ;%{PE}
;FOLD Parameters ;%{h}
;Params IlfProvider=kukaroboter.basistech.inlineforms.movement.old; Kuka.IsGlobalPoint=False; Kuka.PointName=P474; Kuka.BlendingEnabled=False; Kuka.MoveDataName=CPDAT1; Kuka.VelocityPath=2; Kuka.CurrentCDSetIndex=0; Kuka.MovementParameterFieldEnabled=True; IlfCommand=LIN
;ENDFOLD
$BWDSTART = FALSE
LDAT_ACT = LCPDAT474
FDAT_ACT = FP474
BAS(#CP_PARAMS, 2.0)
SET_CD_PARAMS (0)
LIN XP474
;ENDFOLD

;FOLD LIN P475 Vel=2 m/s CPDAT475 Tool[1]:marker Base[0] ;%{PE}
;FOLD Parameters ;%{h}
;Params IlfProvider=kukaroboter.basistech.inlineforms.movement.old; Kuka.IsGlobalPoint=False; Kuka.PointName=P475; Kuka.BlendingEnabled=False; Kuka.MoveDataName=CPDAT1; Kuka.VelocityPath=2; Kuka.CurrentCDSetIndex=0; Kuka.MovementParameterFieldEnabled=True; IlfCommand=LIN
;ENDFOLD
$BWDSTART = FALSE
LDAT_ACT = LCPDAT475
FDAT_ACT = FP475
BAS(#CP_PARAMS, 2.0)
SET_CD_PARAMS (0)
LIN XP475
;ENDFOLD

;FOLD LIN P476 Vel=2 m/s CPDAT476 Tool[1]:marker Base[0] ;%{PE}
;FOLD Parameters ;%{h}
;Params IlfProvider=kukaroboter.basistech.inlineforms.movement.old; Kuka.IsGlobalPoint=False; Kuka.PointName=P476; Kuka.BlendingEnabled=False; Kuka.MoveDataName=CPDAT1; Kuka.VelocityPath=2; Kuka.CurrentCDSetIndex=0; Kuka.MovementParameterFieldEnabled=True; IlfCommand=LIN
;ENDFOLD
$BWDSTART = FALSE
LDAT_ACT = LCPDAT476
FDAT_ACT = FP476
BAS(#CP_PARAMS, 2.0)
SET_CD_PARAMS (0)
LIN XP476
;ENDFOLD

;FOLD LIN P477 Vel=2 m/s CPDAT477 Tool[1]:marker Base[0] ;%{PE}
;FOLD Parameters ;%{h}
;Params IlfProvider=kukaroboter.basistech.inlineforms.movement.old; Kuka.IsGlobalPoint=False; Kuka.PointName=P477; Kuka.BlendingEnabled=False; Kuka.MoveDataName=CPDAT1; Kuka.VelocityPath=2; Kuka.CurrentCDSetIndex=0; Kuka.MovementParameterFieldEnabled=True; IlfCommand=LIN
;ENDFOLD
$BWDSTART = FALSE
LDAT_ACT = LCPDAT477
FDAT_ACT = FP477
BAS(#CP_PARAMS, 2.0)
SET_CD_PARAMS (0)
LIN XP477
;ENDFOLD

;FOLD LIN P478 Vel=2 m/s CPDAT478 Tool[1]:marker Base[0] ;%{PE}
;FOLD Parameters ;%{h}
;Params IlfProvider=kukaroboter.basistech.inlineforms.movement.old; Kuka.IsGlobalPoint=False; Kuka.PointName=P478; Kuka.BlendingEnabled=False; Kuka.MoveDataName=CPDAT1; Kuka.VelocityPath=2; Kuka.CurrentCDSetIndex=0; Kuka.MovementParameterFieldEnabled=True; IlfCommand=LIN
;ENDFOLD
$BWDSTART = FALSE
LDAT_ACT = LCPDAT478
FDAT_ACT = FP478
BAS(#CP_PARAMS, 2.0)
SET_CD_PARAMS (0)
LIN XP478
;ENDFOLD

;FOLD LIN P479 Vel=2 m/s CPDAT479 Tool[1]:marker Base[0] ;%{PE}
;FOLD Parameters ;%{h}
;Params IlfProvider=kukaroboter.basistech.inlineforms.movement.old; Kuka.IsGlobalPoint=False; Kuka.PointName=P479; Kuka.BlendingEnabled=False; Kuka.MoveDataName=CPDAT1; Kuka.VelocityPath=2; Kuka.CurrentCDSetIndex=0; Kuka.MovementParameterFieldEnabled=True; IlfCommand=LIN
;ENDFOLD
$BWDSTART = FALSE
LDAT_ACT = LCPDAT479
FDAT_ACT = FP479
BAS(#CP_PARAMS, 2.0)
SET_CD_PARAMS (0)
LIN XP479
;ENDFOLD

;FOLD LIN P480 Vel=2 m/s CPDAT480 Tool[1]:marker Base[0] ;%{PE}
;FOLD Parameters ;%{h}
;Params IlfProvider=kukaroboter.basistech.inlineforms.movement.old; Kuka.IsGlobalPoint=False; Kuka.PointName=P480; Kuka.BlendingEnabled=False; Kuka.MoveDataName=CPDAT1; Kuka.VelocityPath=2; Kuka.CurrentCDSetIndex=0; Kuka.MovementParameterFieldEnabled=True; IlfCommand=LIN
;ENDFOLD
$BWDSTART = FALSE
LDAT_ACT = LCPDAT480
FDAT_ACT = FP480
BAS(#CP_PARAMS, 2.0)
SET_CD_PARAMS (0)
LIN XP480
;ENDFOLD

;FOLD LIN P481 Vel=2 m/s CPDAT481 Tool[1]:marker Base[0] ;%{PE}
;FOLD Parameters ;%{h}
;Params IlfProvider=kukaroboter.basistech.inlineforms.movement.old; Kuka.IsGlobalPoint=False; Kuka.PointName=P481; Kuka.BlendingEnabled=False; Kuka.MoveDataName=CPDAT1; Kuka.VelocityPath=2; Kuka.CurrentCDSetIndex=0; Kuka.MovementParameterFieldEnabled=True; IlfCommand=LIN
;ENDFOLD
$BWDSTART = FALSE
LDAT_ACT = LCPDAT481
FDAT_ACT = FP481
BAS(#CP_PARAMS, 2.0)
SET_CD_PARAMS (0)
LIN XP481
;ENDFOLD

;FOLD LIN P482 Vel=2 m/s CPDAT482 Tool[1]:marker Base[0] ;%{PE}
;FOLD Parameters ;%{h}
;Params IlfProvider=kukaroboter.basistech.inlineforms.movement.old; Kuka.IsGlobalPoint=False; Kuka.PointName=P482; Kuka.BlendingEnabled=False; Kuka.MoveDataName=CPDAT1; Kuka.VelocityPath=2; Kuka.CurrentCDSetIndex=0; Kuka.MovementParameterFieldEnabled=True; IlfCommand=LIN
;ENDFOLD
$BWDSTART = FALSE
LDAT_ACT = LCPDAT482
FDAT_ACT = FP482
BAS(#CP_PARAMS, 2.0)
SET_CD_PARAMS (0)
LIN XP482
;ENDFOLD

;FOLD LIN P483 Vel=2 m/s CPDAT483 Tool[1]:marker Base[0] ;%{PE}
;FOLD Parameters ;%{h}
;Params IlfProvider=kukaroboter.basistech.inlineforms.movement.old; Kuka.IsGlobalPoint=False; Kuka.PointName=P483; Kuka.BlendingEnabled=False; Kuka.MoveDataName=CPDAT1; Kuka.VelocityPath=2; Kuka.CurrentCDSetIndex=0; Kuka.MovementParameterFieldEnabled=True; IlfCommand=LIN
;ENDFOLD
$BWDSTART = FALSE
LDAT_ACT = LCPDAT483
FDAT_ACT = FP483
BAS(#CP_PARAMS, 2.0)
SET_CD_PARAMS (0)
LIN XP483
;ENDFOLD

;FOLD LIN P484 Vel=2 m/s CPDAT484 Tool[1]:marker Base[0] ;%{PE}
;FOLD Parameters ;%{h}
;Params IlfProvider=kukaroboter.basistech.inlineforms.movement.old; Kuka.IsGlobalPoint=False; Kuka.PointName=P484; Kuka.BlendingEnabled=False; Kuka.MoveDataName=CPDAT1; Kuka.VelocityPath=2; Kuka.CurrentCDSetIndex=0; Kuka.MovementParameterFieldEnabled=True; IlfCommand=LIN
;ENDFOLD
$BWDSTART = FALSE
LDAT_ACT = LCPDAT484
FDAT_ACT = FP484
BAS(#CP_PARAMS, 2.0)
SET_CD_PARAMS (0)
LIN XP484
;ENDFOLD

;FOLD LIN P485 Vel=2 m/s CPDAT485 Tool[1]:marker Base[0] ;%{PE}
;FOLD Parameters ;%{h}
;Params IlfProvider=kukaroboter.basistech.inlineforms.movement.old; Kuka.IsGlobalPoint=False; Kuka.PointName=P485; Kuka.BlendingEnabled=False; Kuka.MoveDataName=CPDAT1; Kuka.VelocityPath=2; Kuka.CurrentCDSetIndex=0; Kuka.MovementParameterFieldEnabled=True; IlfCommand=LIN
;ENDFOLD
$BWDSTART = FALSE
LDAT_ACT = LCPDAT485
FDAT_ACT = FP485
BAS(#CP_PARAMS, 2.0)
SET_CD_PARAMS (0)
LIN XP485
;ENDFOLD

;FOLD LIN P486 Vel=2 m/s CPDAT486 Tool[1]:marker Base[0] ;%{PE}
;FOLD Parameters ;%{h}
;Params IlfProvider=kukaroboter.basistech.inlineforms.movement.old; Kuka.IsGlobalPoint=False; Kuka.PointName=P486; Kuka.BlendingEnabled=False; Kuka.MoveDataName=CPDAT1; Kuka.VelocityPath=2; Kuka.CurrentCDSetIndex=0; Kuka.MovementParameterFieldEnabled=True; IlfCommand=LIN
;ENDFOLD
$BWDSTART = FALSE
LDAT_ACT = LCPDAT486
FDAT_ACT = FP486
BAS(#CP_PARAMS, 2.0)
SET_CD_PARAMS (0)
LIN XP486
;ENDFOLD

;FOLD LIN P487 Vel=2 m/s CPDAT487 Tool[1]:marker Base[0] ;%{PE}
;FOLD Parameters ;%{h}
;Params IlfProvider=kukaroboter.basistech.inlineforms.movement.old; Kuka.IsGlobalPoint=False; Kuka.PointName=P487; Kuka.BlendingEnabled=False; Kuka.MoveDataName=CPDAT1; Kuka.VelocityPath=2; Kuka.CurrentCDSetIndex=0; Kuka.MovementParameterFieldEnabled=True; IlfCommand=LIN
;ENDFOLD
$BWDSTART = FALSE
LDAT_ACT = LCPDAT487
FDAT_ACT = FP487
BAS(#CP_PARAMS, 2.0)
SET_CD_PARAMS (0)
LIN XP487
;ENDFOLD

;FOLD LIN P488 Vel=2 m/s CPDAT488 Tool[1]:marker Base[0] ;%{PE}
;FOLD Parameters ;%{h}
;Params IlfProvider=kukaroboter.basistech.inlineforms.movement.old; Kuka.IsGlobalPoint=False; Kuka.PointName=P488; Kuka.BlendingEnabled=False; Kuka.MoveDataName=CPDAT1; Kuka.VelocityPath=2; Kuka.CurrentCDSetIndex=0; Kuka.MovementParameterFieldEnabled=True; IlfCommand=LIN
;ENDFOLD
$BWDSTART = FALSE
LDAT_ACT = LCPDAT488
FDAT_ACT = FP488
BAS(#CP_PARAMS, 2.0)
SET_CD_PARAMS (0)
LIN XP488
;ENDFOLD

;FOLD LIN P489 Vel=2 m/s CPDAT489 Tool[1]:marker Base[0] ;%{PE}
;FOLD Parameters ;%{h}
;Params IlfProvider=kukaroboter.basistech.inlineforms.movement.old; Kuka.IsGlobalPoint=False; Kuka.PointName=P489; Kuka.BlendingEnabled=False; Kuka.MoveDataName=CPDAT1; Kuka.VelocityPath=2; Kuka.CurrentCDSetIndex=0; Kuka.MovementParameterFieldEnabled=True; IlfCommand=LIN
;ENDFOLD
$BWDSTART = FALSE
LDAT_ACT = LCPDAT489
FDAT_ACT = FP489
BAS(#CP_PARAMS, 2.0)
SET_CD_PARAMS (0)
LIN XP489
;ENDFOLD

;FOLD LIN P490 Vel=2 m/s CPDAT490 Tool[1]:marker Base[0] ;%{PE}
;FOLD Parameters ;%{h}
;Params IlfProvider=kukaroboter.basistech.inlineforms.movement.old; Kuka.IsGlobalPoint=False; Kuka.PointName=P490; Kuka.BlendingEnabled=False; Kuka.MoveDataName=CPDAT1; Kuka.VelocityPath=2; Kuka.CurrentCDSetIndex=0; Kuka.MovementParameterFieldEnabled=True; IlfCommand=LIN
;ENDFOLD
$BWDSTART = FALSE
LDAT_ACT = LCPDAT490
FDAT_ACT = FP490
BAS(#CP_PARAMS, 2.0)
SET_CD_PARAMS (0)
LIN XP490
;ENDFOLD

;FOLD LIN P491 Vel=2 m/s CPDAT491 Tool[1]:marker Base[0] ;%{PE}
;FOLD Parameters ;%{h}
;Params IlfProvider=kukaroboter.basistech.inlineforms.movement.old; Kuka.IsGlobalPoint=False; Kuka.PointName=P491; Kuka.BlendingEnabled=False; Kuka.MoveDataName=CPDAT1; Kuka.VelocityPath=2; Kuka.CurrentCDSetIndex=0; Kuka.MovementParameterFieldEnabled=True; IlfCommand=LIN
;ENDFOLD
$BWDSTART = FALSE
LDAT_ACT = LCPDAT491
FDAT_ACT = FP491
BAS(#CP_PARAMS, 2.0)
SET_CD_PARAMS (0)
LIN XP491
;ENDFOLD

;FOLD LIN P492 Vel=2 m/s CPDAT492 Tool[1]:marker Base[0] ;%{PE}
;FOLD Parameters ;%{h}
;Params IlfProvider=kukaroboter.basistech.inlineforms.movement.old; Kuka.IsGlobalPoint=False; Kuka.PointName=P492; Kuka.BlendingEnabled=False; Kuka.MoveDataName=CPDAT1; Kuka.VelocityPath=2; Kuka.CurrentCDSetIndex=0; Kuka.MovementParameterFieldEnabled=True; IlfCommand=LIN
;ENDFOLD
$BWDSTART = FALSE
LDAT_ACT = LCPDAT492
FDAT_ACT = FP492
BAS(#CP_PARAMS, 2.0)
SET_CD_PARAMS (0)
LIN XP492
;ENDFOLD

;FOLD LIN P493 Vel=2 m/s CPDAT493 Tool[1]:marker Base[0] ;%{PE}
;FOLD Parameters ;%{h}
;Params IlfProvider=kukaroboter.basistech.inlineforms.movement.old; Kuka.IsGlobalPoint=False; Kuka.PointName=P493; Kuka.BlendingEnabled=False; Kuka.MoveDataName=CPDAT1; Kuka.VelocityPath=2; Kuka.CurrentCDSetIndex=0; Kuka.MovementParameterFieldEnabled=True; IlfCommand=LIN
;ENDFOLD
$BWDSTART = FALSE
LDAT_ACT = LCPDAT493
FDAT_ACT = FP493
BAS(#CP_PARAMS, 2.0)
SET_CD_PARAMS (0)
LIN XP493
;ENDFOLD

;FOLD LIN P494 Vel=2 m/s CPDAT494 Tool[1]:marker Base[0] ;%{PE}
;FOLD Parameters ;%{h}
;Params IlfProvider=kukaroboter.basistech.inlineforms.movement.old; Kuka.IsGlobalPoint=False; Kuka.PointName=P494; Kuka.BlendingEnabled=False; Kuka.MoveDataName=CPDAT1; Kuka.VelocityPath=2; Kuka.CurrentCDSetIndex=0; Kuka.MovementParameterFieldEnabled=True; IlfCommand=LIN
;ENDFOLD
$BWDSTART = FALSE
LDAT_ACT = LCPDAT494
FDAT_ACT = FP494
BAS(#CP_PARAMS, 2.0)
SET_CD_PARAMS (0)
LIN XP494
;ENDFOLD

;FOLD LIN P495 Vel=2 m/s CPDAT495 Tool[1]:marker Base[0] ;%{PE}
;FOLD Parameters ;%{h}
;Params IlfProvider=kukaroboter.basistech.inlineforms.movement.old; Kuka.IsGlobalPoint=False; Kuka.PointName=P495; Kuka.BlendingEnabled=False; Kuka.MoveDataName=CPDAT1; Kuka.VelocityPath=2; Kuka.CurrentCDSetIndex=0; Kuka.MovementParameterFieldEnabled=True; IlfCommand=LIN
;ENDFOLD
$BWDSTART = FALSE
LDAT_ACT = LCPDAT495
FDAT_ACT = FP495
BAS(#CP_PARAMS, 2.0)
SET_CD_PARAMS (0)
LIN XP495
;ENDFOLD

;FOLD LIN P496 Vel=2 m/s CPDAT496 Tool[1]:marker Base[0] ;%{PE}
;FOLD Parameters ;%{h}
;Params IlfProvider=kukaroboter.basistech.inlineforms.movement.old; Kuka.IsGlobalPoint=False; Kuka.PointName=P496; Kuka.BlendingEnabled=False; Kuka.MoveDataName=CPDAT1; Kuka.VelocityPath=2; Kuka.CurrentCDSetIndex=0; Kuka.MovementParameterFieldEnabled=True; IlfCommand=LIN
;ENDFOLD
$BWDSTART = FALSE
LDAT_ACT = LCPDAT496
FDAT_ACT = FP496
BAS(#CP_PARAMS, 2.0)
SET_CD_PARAMS (0)
LIN XP496
;ENDFOLD

;FOLD LIN P497 Vel=2 m/s CPDAT497 Tool[1]:marker Base[0] ;%{PE}
;FOLD Parameters ;%{h}
;Params IlfProvider=kukaroboter.basistech.inlineforms.movement.old; Kuka.IsGlobalPoint=False; Kuka.PointName=P497; Kuka.BlendingEnabled=False; Kuka.MoveDataName=CPDAT1; Kuka.VelocityPath=2; Kuka.CurrentCDSetIndex=0; Kuka.MovementParameterFieldEnabled=True; IlfCommand=LIN
;ENDFOLD
$BWDSTART = FALSE
LDAT_ACT = LCPDAT497
FDAT_ACT = FP497
BAS(#CP_PARAMS, 2.0)
SET_CD_PARAMS (0)
LIN XP497
;ENDFOLD

;FOLD LIN P498 Vel=2 m/s CPDAT498 Tool[1]:marker Base[0] ;%{PE}
;FOLD Parameters ;%{h}
;Params IlfProvider=kukaroboter.basistech.inlineforms.movement.old; Kuka.IsGlobalPoint=False; Kuka.PointName=P498; Kuka.BlendingEnabled=False; Kuka.MoveDataName=CPDAT1; Kuka.VelocityPath=2; Kuka.CurrentCDSetIndex=0; Kuka.MovementParameterFieldEnabled=True; IlfCommand=LIN
;ENDFOLD
$BWDSTART = FALSE
LDAT_ACT = LCPDAT498
FDAT_ACT = FP498
BAS(#CP_PARAMS, 2.0)
SET_CD_PARAMS (0)
LIN XP498
;ENDFOLD

;FOLD LIN P499 Vel=2 m/s CPDAT499 Tool[1]:marker Base[0] ;%{PE}
;FOLD Parameters ;%{h}
;Params IlfProvider=kukaroboter.basistech.inlineforms.movement.old; Kuka.IsGlobalPoint=False; Kuka.PointName=P499; Kuka.BlendingEnabled=False; Kuka.MoveDataName=CPDAT1; Kuka.VelocityPath=2; Kuka.CurrentCDSetIndex=0; Kuka.MovementParameterFieldEnabled=True; IlfCommand=LIN
;ENDFOLD
$BWDSTART = FALSE
LDAT_ACT = LCPDAT499
FDAT_ACT = FP499
BAS(#CP_PARAMS, 2.0)
SET_CD_PARAMS (0)
LIN XP499
;ENDFOLD

;FOLD LIN P500 Vel=2 m/s CPDAT500 Tool[1]:marker Base[0] ;%{PE}
;FOLD Parameters ;%{h}
;Params IlfProvider=kukaroboter.basistech.inlineforms.movement.old; Kuka.IsGlobalPoint=False; Kuka.PointName=P500; Kuka.BlendingEnabled=False; Kuka.MoveDataName=CPDAT1; Kuka.VelocityPath=2; Kuka.CurrentCDSetIndex=0; Kuka.MovementParameterFieldEnabled=True; IlfCommand=LIN
;ENDFOLD
$BWDSTART = FALSE
LDAT_ACT = LCPDAT500
FDAT_ACT = FP500
BAS(#CP_PARAMS, 2.0)
SET_CD_PARAMS (0)
LIN XP500
;ENDFOLD

;FOLD LIN P501 Vel=2 m/s CPDAT501 Tool[1]:marker Base[0] ;%{PE}
;FOLD Parameters ;%{h}
;Params IlfProvider=kukaroboter.basistech.inlineforms.movement.old; Kuka.IsGlobalPoint=False; Kuka.PointName=P501; Kuka.BlendingEnabled=False; Kuka.MoveDataName=CPDAT1; Kuka.VelocityPath=2; Kuka.CurrentCDSetIndex=0; Kuka.MovementParameterFieldEnabled=True; IlfCommand=LIN
;ENDFOLD
$BWDSTART = FALSE
LDAT_ACT = LCPDAT501
FDAT_ACT = FP501
BAS(#CP_PARAMS, 2.0)
SET_CD_PARAMS (0)
LIN XP501
;ENDFOLD

;FOLD LIN P502 Vel=2 m/s CPDAT502 Tool[1]:marker Base[0] ;%{PE}
;FOLD Parameters ;%{h}
;Params IlfProvider=kukaroboter.basistech.inlineforms.movement.old; Kuka.IsGlobalPoint=False; Kuka.PointName=P502; Kuka.BlendingEnabled=False; Kuka.MoveDataName=CPDAT1; Kuka.VelocityPath=2; Kuka.CurrentCDSetIndex=0; Kuka.MovementParameterFieldEnabled=True; IlfCommand=LIN
;ENDFOLD
$BWDSTART = FALSE
LDAT_ACT = LCPDAT502
FDAT_ACT = FP502
BAS(#CP_PARAMS, 2.0)
SET_CD_PARAMS (0)
LIN XP502
;ENDFOLD

;FOLD LIN P503 Vel=2 m/s CPDAT503 Tool[1]:marker Base[0] ;%{PE}
;FOLD Parameters ;%{h}
;Params IlfProvider=kukaroboter.basistech.inlineforms.movement.old; Kuka.IsGlobalPoint=False; Kuka.PointName=P503; Kuka.BlendingEnabled=False; Kuka.MoveDataName=CPDAT1; Kuka.VelocityPath=2; Kuka.CurrentCDSetIndex=0; Kuka.MovementParameterFieldEnabled=True; IlfCommand=LIN
;ENDFOLD
$BWDSTART = FALSE
LDAT_ACT = LCPDAT503
FDAT_ACT = FP503
BAS(#CP_PARAMS, 2.0)
SET_CD_PARAMS (0)
LIN XP503
;ENDFOLD

;FOLD LIN P504 Vel=2 m/s CPDAT504 Tool[1]:marker Base[0] ;%{PE}
;FOLD Parameters ;%{h}
;Params IlfProvider=kukaroboter.basistech.inlineforms.movement.old; Kuka.IsGlobalPoint=False; Kuka.PointName=P504; Kuka.BlendingEnabled=False; Kuka.MoveDataName=CPDAT1; Kuka.VelocityPath=2; Kuka.CurrentCDSetIndex=0; Kuka.MovementParameterFieldEnabled=True; IlfCommand=LIN
;ENDFOLD
$BWDSTART = FALSE
LDAT_ACT = LCPDAT504
FDAT_ACT = FP504
BAS(#CP_PARAMS, 2.0)
SET_CD_PARAMS (0)
LIN XP504
;ENDFOLD

;FOLD LIN P505 Vel=2 m/s CPDAT505 Tool[1]:marker Base[0] ;%{PE}
;FOLD Parameters ;%{h}
;Params IlfProvider=kukaroboter.basistech.inlineforms.movement.old; Kuka.IsGlobalPoint=False; Kuka.PointName=P505; Kuka.BlendingEnabled=False; Kuka.MoveDataName=CPDAT1; Kuka.VelocityPath=2; Kuka.CurrentCDSetIndex=0; Kuka.MovementParameterFieldEnabled=True; IlfCommand=LIN
;ENDFOLD
$BWDSTART = FALSE
LDAT_ACT = LCPDAT505
FDAT_ACT = FP505
BAS(#CP_PARAMS, 2.0)
SET_CD_PARAMS (0)
LIN XP505
;ENDFOLD

;FOLD LIN P506 Vel=2 m/s CPDAT506 Tool[1]:marker Base[0] ;%{PE}
;FOLD Parameters ;%{h}
;Params IlfProvider=kukaroboter.basistech.inlineforms.movement.old; Kuka.IsGlobalPoint=False; Kuka.PointName=P506; Kuka.BlendingEnabled=False; Kuka.MoveDataName=CPDAT1; Kuka.VelocityPath=2; Kuka.CurrentCDSetIndex=0; Kuka.MovementParameterFieldEnabled=True; IlfCommand=LIN
;ENDFOLD
$BWDSTART = FALSE
LDAT_ACT = LCPDAT506
FDAT_ACT = FP506
BAS(#CP_PARAMS, 2.0)
SET_CD_PARAMS (0)
LIN XP506
;ENDFOLD

;FOLD LIN P507 Vel=2 m/s CPDAT507 Tool[1]:marker Base[0] ;%{PE}
;FOLD Parameters ;%{h}
;Params IlfProvider=kukaroboter.basistech.inlineforms.movement.old; Kuka.IsGlobalPoint=False; Kuka.PointName=P507; Kuka.BlendingEnabled=False; Kuka.MoveDataName=CPDAT1; Kuka.VelocityPath=2; Kuka.CurrentCDSetIndex=0; Kuka.MovementParameterFieldEnabled=True; IlfCommand=LIN
;ENDFOLD
$BWDSTART = FALSE
LDAT_ACT = LCPDAT507
FDAT_ACT = FP507
BAS(#CP_PARAMS, 2.0)
SET_CD_PARAMS (0)
LIN XP507
;ENDFOLD

;FOLD LIN P508 Vel=2 m/s CPDAT508 Tool[1]:marker Base[0] ;%{PE}
;FOLD Parameters ;%{h}
;Params IlfProvider=kukaroboter.basistech.inlineforms.movement.old; Kuka.IsGlobalPoint=False; Kuka.PointName=P508; Kuka.BlendingEnabled=False; Kuka.MoveDataName=CPDAT1; Kuka.VelocityPath=2; Kuka.CurrentCDSetIndex=0; Kuka.MovementParameterFieldEnabled=True; IlfCommand=LIN
;ENDFOLD
$BWDSTART = FALSE
LDAT_ACT = LCPDAT508
FDAT_ACT = FP508
BAS(#CP_PARAMS, 2.0)
SET_CD_PARAMS (0)
LIN XP508
;ENDFOLD

;FOLD LIN P509 Vel=2 m/s CPDAT509 Tool[1]:marker Base[0] ;%{PE}
;FOLD Parameters ;%{h}
;Params IlfProvider=kukaroboter.basistech.inlineforms.movement.old; Kuka.IsGlobalPoint=False; Kuka.PointName=P509; Kuka.BlendingEnabled=False; Kuka.MoveDataName=CPDAT1; Kuka.VelocityPath=2; Kuka.CurrentCDSetIndex=0; Kuka.MovementParameterFieldEnabled=True; IlfCommand=LIN
;ENDFOLD
$BWDSTART = FALSE
LDAT_ACT = LCPDAT509
FDAT_ACT = FP509
BAS(#CP_PARAMS, 2.0)
SET_CD_PARAMS (0)
LIN XP509
;ENDFOLD

;FOLD LIN P510 Vel=2 m/s CPDAT510 Tool[1]:marker Base[0] ;%{PE}
;FOLD Parameters ;%{h}
;Params IlfProvider=kukaroboter.basistech.inlineforms.movement.old; Kuka.IsGlobalPoint=False; Kuka.PointName=P510; Kuka.BlendingEnabled=False; Kuka.MoveDataName=CPDAT1; Kuka.VelocityPath=2; Kuka.CurrentCDSetIndex=0; Kuka.MovementParameterFieldEnabled=True; IlfCommand=LIN
;ENDFOLD
$BWDSTART = FALSE
LDAT_ACT = LCPDAT510
FDAT_ACT = FP510
BAS(#CP_PARAMS, 2.0)
SET_CD_PARAMS (0)
LIN XP510
;ENDFOLD

;FOLD LIN P511 Vel=2 m/s CPDAT511 Tool[1]:marker Base[0] ;%{PE}
;FOLD Parameters ;%{h}
;Params IlfProvider=kukaroboter.basistech.inlineforms.movement.old; Kuka.IsGlobalPoint=False; Kuka.PointName=P511; Kuka.BlendingEnabled=False; Kuka.MoveDataName=CPDAT1; Kuka.VelocityPath=2; Kuka.CurrentCDSetIndex=0; Kuka.MovementParameterFieldEnabled=True; IlfCommand=LIN
;ENDFOLD
$BWDSTART = FALSE
LDAT_ACT = LCPDAT511
FDAT_ACT = FP511
BAS(#CP_PARAMS, 2.0)
SET_CD_PARAMS (0)
LIN XP511
;ENDFOLD

;FOLD LIN P512 Vel=2 m/s CPDAT512 Tool[1]:marker Base[0] ;%{PE}
;FOLD Parameters ;%{h}
;Params IlfProvider=kukaroboter.basistech.inlineforms.movement.old; Kuka.IsGlobalPoint=False; Kuka.PointName=P512; Kuka.BlendingEnabled=False; Kuka.MoveDataName=CPDAT1; Kuka.VelocityPath=2; Kuka.CurrentCDSetIndex=0; Kuka.MovementParameterFieldEnabled=True; IlfCommand=LIN
;ENDFOLD
$BWDSTART = FALSE
LDAT_ACT = LCPDAT512
FDAT_ACT = FP512
BAS(#CP_PARAMS, 2.0)
SET_CD_PARAMS (0)
LIN XP512
;ENDFOLD

;FOLD LIN P513 Vel=2 m/s CPDAT513 Tool[1]:marker Base[0] ;%{PE}
;FOLD Parameters ;%{h}
;Params IlfProvider=kukaroboter.basistech.inlineforms.movement.old; Kuka.IsGlobalPoint=False; Kuka.PointName=P513; Kuka.BlendingEnabled=False; Kuka.MoveDataName=CPDAT1; Kuka.VelocityPath=2; Kuka.CurrentCDSetIndex=0; Kuka.MovementParameterFieldEnabled=True; IlfCommand=LIN
;ENDFOLD
$BWDSTART = FALSE
LDAT_ACT = LCPDAT513
FDAT_ACT = FP513
BAS(#CP_PARAMS, 2.0)
SET_CD_PARAMS (0)
LIN XP513
;ENDFOLD

;FOLD LIN P514 Vel=2 m/s CPDAT514 Tool[1]:marker Base[0] ;%{PE}
;FOLD Parameters ;%{h}
;Params IlfProvider=kukaroboter.basistech.inlineforms.movement.old; Kuka.IsGlobalPoint=False; Kuka.PointName=P514; Kuka.BlendingEnabled=False; Kuka.MoveDataName=CPDAT1; Kuka.VelocityPath=2; Kuka.CurrentCDSetIndex=0; Kuka.MovementParameterFieldEnabled=True; IlfCommand=LIN
;ENDFOLD
$BWDSTART = FALSE
LDAT_ACT = LCPDAT514
FDAT_ACT = FP514
BAS(#CP_PARAMS, 2.0)
SET_CD_PARAMS (0)
LIN XP514
;ENDFOLD

;FOLD LIN P515 Vel=2 m/s CPDAT515 Tool[1]:marker Base[0] ;%{PE}
;FOLD Parameters ;%{h}
;Params IlfProvider=kukaroboter.basistech.inlineforms.movement.old; Kuka.IsGlobalPoint=False; Kuka.PointName=P515; Kuka.BlendingEnabled=False; Kuka.MoveDataName=CPDAT1; Kuka.VelocityPath=2; Kuka.CurrentCDSetIndex=0; Kuka.MovementParameterFieldEnabled=True; IlfCommand=LIN
;ENDFOLD
$BWDSTART = FALSE
LDAT_ACT = LCPDAT515
FDAT_ACT = FP515
BAS(#CP_PARAMS, 2.0)
SET_CD_PARAMS (0)
LIN XP515
;ENDFOLD

;FOLD LIN P516 Vel=2 m/s CPDAT516 Tool[1]:marker Base[0] ;%{PE}
;FOLD Parameters ;%{h}
;Params IlfProvider=kukaroboter.basistech.inlineforms.movement.old; Kuka.IsGlobalPoint=False; Kuka.PointName=P516; Kuka.BlendingEnabled=False; Kuka.MoveDataName=CPDAT1; Kuka.VelocityPath=2; Kuka.CurrentCDSetIndex=0; Kuka.MovementParameterFieldEnabled=True; IlfCommand=LIN
;ENDFOLD
$BWDSTART = FALSE
LDAT_ACT = LCPDAT516
FDAT_ACT = FP516
BAS(#CP_PARAMS, 2.0)
SET_CD_PARAMS (0)
LIN XP516
;ENDFOLD

;FOLD LIN P517 Vel=2 m/s CPDAT517 Tool[1]:marker Base[0] ;%{PE}
;FOLD Parameters ;%{h}
;Params IlfProvider=kukaroboter.basistech.inlineforms.movement.old; Kuka.IsGlobalPoint=False; Kuka.PointName=P517; Kuka.BlendingEnabled=False; Kuka.MoveDataName=CPDAT1; Kuka.VelocityPath=2; Kuka.CurrentCDSetIndex=0; Kuka.MovementParameterFieldEnabled=True; IlfCommand=LIN
;ENDFOLD
$BWDSTART = FALSE
LDAT_ACT = LCPDAT517
FDAT_ACT = FP517
BAS(#CP_PARAMS, 2.0)
SET_CD_PARAMS (0)
LIN XP517
;ENDFOLD

;FOLD LIN P518 Vel=2 m/s CPDAT518 Tool[1]:marker Base[0] ;%{PE}
;FOLD Parameters ;%{h}
;Params IlfProvider=kukaroboter.basistech.inlineforms.movement.old; Kuka.IsGlobalPoint=False; Kuka.PointName=P518; Kuka.BlendingEnabled=False; Kuka.MoveDataName=CPDAT1; Kuka.VelocityPath=2; Kuka.CurrentCDSetIndex=0; Kuka.MovementParameterFieldEnabled=True; IlfCommand=LIN
;ENDFOLD
$BWDSTART = FALSE
LDAT_ACT = LCPDAT518
FDAT_ACT = FP518
BAS(#CP_PARAMS, 2.0)
SET_CD_PARAMS (0)
LIN XP518
;ENDFOLD

;FOLD LIN P519 Vel=2 m/s CPDAT519 Tool[1]:marker Base[0] ;%{PE}
;FOLD Parameters ;%{h}
;Params IlfProvider=kukaroboter.basistech.inlineforms.movement.old; Kuka.IsGlobalPoint=False; Kuka.PointName=P519; Kuka.BlendingEnabled=False; Kuka.MoveDataName=CPDAT1; Kuka.VelocityPath=2; Kuka.CurrentCDSetIndex=0; Kuka.MovementParameterFieldEnabled=True; IlfCommand=LIN
;ENDFOLD
$BWDSTART = FALSE
LDAT_ACT = LCPDAT519
FDAT_ACT = FP519
BAS(#CP_PARAMS, 2.0)
SET_CD_PARAMS (0)
LIN XP519
;ENDFOLD

;FOLD LIN P520 Vel=2 m/s CPDAT520 Tool[1]:marker Base[0] ;%{PE}
;FOLD Parameters ;%{h}
;Params IlfProvider=kukaroboter.basistech.inlineforms.movement.old; Kuka.IsGlobalPoint=False; Kuka.PointName=P520; Kuka.BlendingEnabled=False; Kuka.MoveDataName=CPDAT1; Kuka.VelocityPath=2; Kuka.CurrentCDSetIndex=0; Kuka.MovementParameterFieldEnabled=True; IlfCommand=LIN
;ENDFOLD
$BWDSTART = FALSE
LDAT_ACT = LCPDAT520
FDAT_ACT = FP520
BAS(#CP_PARAMS, 2.0)
SET_CD_PARAMS (0)
LIN XP520
;ENDFOLD

;FOLD LIN P521 Vel=2 m/s CPDAT521 Tool[1]:marker Base[0] ;%{PE}
;FOLD Parameters ;%{h}
;Params IlfProvider=kukaroboter.basistech.inlineforms.movement.old; Kuka.IsGlobalPoint=False; Kuka.PointName=P521; Kuka.BlendingEnabled=False; Kuka.MoveDataName=CPDAT1; Kuka.VelocityPath=2; Kuka.CurrentCDSetIndex=0; Kuka.MovementParameterFieldEnabled=True; IlfCommand=LIN
;ENDFOLD
$BWDSTART = FALSE
LDAT_ACT = LCPDAT521
FDAT_ACT = FP521
BAS(#CP_PARAMS, 2.0)
SET_CD_PARAMS (0)
LIN XP521
;ENDFOLD

;FOLD LIN P522 Vel=2 m/s CPDAT522 Tool[1]:marker Base[0] ;%{PE}
;FOLD Parameters ;%{h}
;Params IlfProvider=kukaroboter.basistech.inlineforms.movement.old; Kuka.IsGlobalPoint=False; Kuka.PointName=P522; Kuka.BlendingEnabled=False; Kuka.MoveDataName=CPDAT1; Kuka.VelocityPath=2; Kuka.CurrentCDSetIndex=0; Kuka.MovementParameterFieldEnabled=True; IlfCommand=LIN
;ENDFOLD
$BWDSTART = FALSE
LDAT_ACT = LCPDAT522
FDAT_ACT = FP522
BAS(#CP_PARAMS, 2.0)
SET_CD_PARAMS (0)
LIN XP522
;ENDFOLD

;FOLD LIN P523 Vel=2 m/s CPDAT523 Tool[1]:marker Base[0] ;%{PE}
;FOLD Parameters ;%{h}
;Params IlfProvider=kukaroboter.basistech.inlineforms.movement.old; Kuka.IsGlobalPoint=False; Kuka.PointName=P523; Kuka.BlendingEnabled=False; Kuka.MoveDataName=CPDAT1; Kuka.VelocityPath=2; Kuka.CurrentCDSetIndex=0; Kuka.MovementParameterFieldEnabled=True; IlfCommand=LIN
;ENDFOLD
$BWDSTART = FALSE
LDAT_ACT = LCPDAT523
FDAT_ACT = FP523
BAS(#CP_PARAMS, 2.0)
SET_CD_PARAMS (0)
LIN XP523
;ENDFOLD

;FOLD LIN P524 Vel=2 m/s CPDAT524 Tool[1]:marker Base[0] ;%{PE}
;FOLD Parameters ;%{h}
;Params IlfProvider=kukaroboter.basistech.inlineforms.movement.old; Kuka.IsGlobalPoint=False; Kuka.PointName=P524; Kuka.BlendingEnabled=False; Kuka.MoveDataName=CPDAT1; Kuka.VelocityPath=2; Kuka.CurrentCDSetIndex=0; Kuka.MovementParameterFieldEnabled=True; IlfCommand=LIN
;ENDFOLD
$BWDSTART = FALSE
LDAT_ACT = LCPDAT524
FDAT_ACT = FP524
BAS(#CP_PARAMS, 2.0)
SET_CD_PARAMS (0)
LIN XP524
;ENDFOLD

;FOLD LIN P525 Vel=2 m/s CPDAT525 Tool[1]:marker Base[0] ;%{PE}
;FOLD Parameters ;%{h}
;Params IlfProvider=kukaroboter.basistech.inlineforms.movement.old; Kuka.IsGlobalPoint=False; Kuka.PointName=P525; Kuka.BlendingEnabled=False; Kuka.MoveDataName=CPDAT1; Kuka.VelocityPath=2; Kuka.CurrentCDSetIndex=0; Kuka.MovementParameterFieldEnabled=True; IlfCommand=LIN
;ENDFOLD
$BWDSTART = FALSE
LDAT_ACT = LCPDAT525
FDAT_ACT = FP525
BAS(#CP_PARAMS, 2.0)
SET_CD_PARAMS (0)
LIN XP525
;ENDFOLD

;FOLD LIN P526 Vel=2 m/s CPDAT526 Tool[1]:marker Base[0] ;%{PE}
;FOLD Parameters ;%{h}
;Params IlfProvider=kukaroboter.basistech.inlineforms.movement.old; Kuka.IsGlobalPoint=False; Kuka.PointName=P526; Kuka.BlendingEnabled=False; Kuka.MoveDataName=CPDAT1; Kuka.VelocityPath=2; Kuka.CurrentCDSetIndex=0; Kuka.MovementParameterFieldEnabled=True; IlfCommand=LIN
;ENDFOLD
$BWDSTART = FALSE
LDAT_ACT = LCPDAT526
FDAT_ACT = FP526
BAS(#CP_PARAMS, 2.0)
SET_CD_PARAMS (0)
LIN XP526
;ENDFOLD

;FOLD LIN P527 Vel=2 m/s CPDAT527 Tool[1]:marker Base[0] ;%{PE}
;FOLD Parameters ;%{h}
;Params IlfProvider=kukaroboter.basistech.inlineforms.movement.old; Kuka.IsGlobalPoint=False; Kuka.PointName=P527; Kuka.BlendingEnabled=False; Kuka.MoveDataName=CPDAT1; Kuka.VelocityPath=2; Kuka.CurrentCDSetIndex=0; Kuka.MovementParameterFieldEnabled=True; IlfCommand=LIN
;ENDFOLD
$BWDSTART = FALSE
LDAT_ACT = LCPDAT527
FDAT_ACT = FP527
BAS(#CP_PARAMS, 2.0)
SET_CD_PARAMS (0)
LIN XP527
;ENDFOLD

;FOLD LIN P528 Vel=2 m/s CPDAT528 Tool[1]:marker Base[0] ;%{PE}
;FOLD Parameters ;%{h}
;Params IlfProvider=kukaroboter.basistech.inlineforms.movement.old; Kuka.IsGlobalPoint=False; Kuka.PointName=P528; Kuka.BlendingEnabled=False; Kuka.MoveDataName=CPDAT1; Kuka.VelocityPath=2; Kuka.CurrentCDSetIndex=0; Kuka.MovementParameterFieldEnabled=True; IlfCommand=LIN
;ENDFOLD
$BWDSTART = FALSE
LDAT_ACT = LCPDAT528
FDAT_ACT = FP528
BAS(#CP_PARAMS, 2.0)
SET_CD_PARAMS (0)
LIN XP528
;ENDFOLD

;FOLD LIN P529 Vel=2 m/s CPDAT529 Tool[1]:marker Base[0] ;%{PE}
;FOLD Parameters ;%{h}
;Params IlfProvider=kukaroboter.basistech.inlineforms.movement.old; Kuka.IsGlobalPoint=False; Kuka.PointName=P529; Kuka.BlendingEnabled=False; Kuka.MoveDataName=CPDAT1; Kuka.VelocityPath=2; Kuka.CurrentCDSetIndex=0; Kuka.MovementParameterFieldEnabled=True; IlfCommand=LIN
;ENDFOLD
$BWDSTART = FALSE
LDAT_ACT = LCPDAT529
FDAT_ACT = FP529
BAS(#CP_PARAMS, 2.0)
SET_CD_PARAMS (0)
LIN XP529
;ENDFOLD

;FOLD LIN P530 Vel=2 m/s CPDAT530 Tool[1]:marker Base[0] ;%{PE}
;FOLD Parameters ;%{h}
;Params IlfProvider=kukaroboter.basistech.inlineforms.movement.old; Kuka.IsGlobalPoint=False; Kuka.PointName=P530; Kuka.BlendingEnabled=False; Kuka.MoveDataName=CPDAT1; Kuka.VelocityPath=2; Kuka.CurrentCDSetIndex=0; Kuka.MovementParameterFieldEnabled=True; IlfCommand=LIN
;ENDFOLD
$BWDSTART = FALSE
LDAT_ACT = LCPDAT530
FDAT_ACT = FP530
BAS(#CP_PARAMS, 2.0)
SET_CD_PARAMS (0)
LIN XP530
;ENDFOLD

;FOLD LIN P531 Vel=2 m/s CPDAT531 Tool[1]:marker Base[0] ;%{PE}
;FOLD Parameters ;%{h}
;Params IlfProvider=kukaroboter.basistech.inlineforms.movement.old; Kuka.IsGlobalPoint=False; Kuka.PointName=P531; Kuka.BlendingEnabled=False; Kuka.MoveDataName=CPDAT1; Kuka.VelocityPath=2; Kuka.CurrentCDSetIndex=0; Kuka.MovementParameterFieldEnabled=True; IlfCommand=LIN
;ENDFOLD
$BWDSTART = FALSE
LDAT_ACT = LCPDAT531
FDAT_ACT = FP531
BAS(#CP_PARAMS, 2.0)
SET_CD_PARAMS (0)
LIN XP531
;ENDFOLD

;FOLD LIN P532 Vel=2 m/s CPDAT532 Tool[1]:marker Base[0] ;%{PE}
;FOLD Parameters ;%{h}
;Params IlfProvider=kukaroboter.basistech.inlineforms.movement.old; Kuka.IsGlobalPoint=False; Kuka.PointName=P532; Kuka.BlendingEnabled=False; Kuka.MoveDataName=CPDAT1; Kuka.VelocityPath=2; Kuka.CurrentCDSetIndex=0; Kuka.MovementParameterFieldEnabled=True; IlfCommand=LIN
;ENDFOLD
$BWDSTART = FALSE
LDAT_ACT = LCPDAT532
FDAT_ACT = FP532
BAS(#CP_PARAMS, 2.0)
SET_CD_PARAMS (0)
LIN XP532
;ENDFOLD

;FOLD LIN P533 Vel=2 m/s CPDAT533 Tool[1]:marker Base[0] ;%{PE}
;FOLD Parameters ;%{h}
;Params IlfProvider=kukaroboter.basistech.inlineforms.movement.old; Kuka.IsGlobalPoint=False; Kuka.PointName=P533; Kuka.BlendingEnabled=False; Kuka.MoveDataName=CPDAT1; Kuka.VelocityPath=2; Kuka.CurrentCDSetIndex=0; Kuka.MovementParameterFieldEnabled=True; IlfCommand=LIN
;ENDFOLD
$BWDSTART = FALSE
LDAT_ACT = LCPDAT533
FDAT_ACT = FP533
BAS(#CP_PARAMS, 2.0)
SET_CD_PARAMS (0)
LIN XP533
;ENDFOLD

;FOLD LIN P534 Vel=2 m/s CPDAT534 Tool[1]:marker Base[0] ;%{PE}
;FOLD Parameters ;%{h}
;Params IlfProvider=kukaroboter.basistech.inlineforms.movement.old; Kuka.IsGlobalPoint=False; Kuka.PointName=P534; Kuka.BlendingEnabled=False; Kuka.MoveDataName=CPDAT1; Kuka.VelocityPath=2; Kuka.CurrentCDSetIndex=0; Kuka.MovementParameterFieldEnabled=True; IlfCommand=LIN
;ENDFOLD
$BWDSTART = FALSE
LDAT_ACT = LCPDAT534
FDAT_ACT = FP534
BAS(#CP_PARAMS, 2.0)
SET_CD_PARAMS (0)
LIN XP534
;ENDFOLD

;FOLD LIN P535 Vel=2 m/s CPDAT535 Tool[1]:marker Base[0] ;%{PE}
;FOLD Parameters ;%{h}
;Params IlfProvider=kukaroboter.basistech.inlineforms.movement.old; Kuka.IsGlobalPoint=False; Kuka.PointName=P535; Kuka.BlendingEnabled=False; Kuka.MoveDataName=CPDAT1; Kuka.VelocityPath=2; Kuka.CurrentCDSetIndex=0; Kuka.MovementParameterFieldEnabled=True; IlfCommand=LIN
;ENDFOLD
$BWDSTART = FALSE
LDAT_ACT = LCPDAT535
FDAT_ACT = FP535
BAS(#CP_PARAMS, 2.0)
SET_CD_PARAMS (0)
LIN XP535
;ENDFOLD

;FOLD LIN P536 Vel=2 m/s CPDAT536 Tool[1]:marker Base[0] ;%{PE}
;FOLD Parameters ;%{h}
;Params IlfProvider=kukaroboter.basistech.inlineforms.movement.old; Kuka.IsGlobalPoint=False; Kuka.PointName=P536; Kuka.BlendingEnabled=False; Kuka.MoveDataName=CPDAT1; Kuka.VelocityPath=2; Kuka.CurrentCDSetIndex=0; Kuka.MovementParameterFieldEnabled=True; IlfCommand=LIN
;ENDFOLD
$BWDSTART = FALSE
LDAT_ACT = LCPDAT536
FDAT_ACT = FP536
BAS(#CP_PARAMS, 2.0)
SET_CD_PARAMS (0)
LIN XP536
;ENDFOLD

;FOLD LIN P537 Vel=2 m/s CPDAT537 Tool[1]:marker Base[0] ;%{PE}
;FOLD Parameters ;%{h}
;Params IlfProvider=kukaroboter.basistech.inlineforms.movement.old; Kuka.IsGlobalPoint=False; Kuka.PointName=P537; Kuka.BlendingEnabled=False; Kuka.MoveDataName=CPDAT1; Kuka.VelocityPath=2; Kuka.CurrentCDSetIndex=0; Kuka.MovementParameterFieldEnabled=True; IlfCommand=LIN
;ENDFOLD
$BWDSTART = FALSE
LDAT_ACT = LCPDAT537
FDAT_ACT = FP537
BAS(#CP_PARAMS, 2.0)
SET_CD_PARAMS (0)
LIN XP537
;ENDFOLD

;FOLD LIN P538 Vel=2 m/s CPDAT538 Tool[1]:marker Base[0] ;%{PE}
;FOLD Parameters ;%{h}
;Params IlfProvider=kukaroboter.basistech.inlineforms.movement.old; Kuka.IsGlobalPoint=False; Kuka.PointName=P538; Kuka.BlendingEnabled=False; Kuka.MoveDataName=CPDAT1; Kuka.VelocityPath=2; Kuka.CurrentCDSetIndex=0; Kuka.MovementParameterFieldEnabled=True; IlfCommand=LIN
;ENDFOLD
$BWDSTART = FALSE
LDAT_ACT = LCPDAT538
FDAT_ACT = FP538
BAS(#CP_PARAMS, 2.0)
SET_CD_PARAMS (0)
LIN XP538
;ENDFOLD

;FOLD LIN P539 Vel=2 m/s CPDAT539 Tool[1]:marker Base[0] ;%{PE}
;FOLD Parameters ;%{h}
;Params IlfProvider=kukaroboter.basistech.inlineforms.movement.old; Kuka.IsGlobalPoint=False; Kuka.PointName=P539; Kuka.BlendingEnabled=False; Kuka.MoveDataName=CPDAT1; Kuka.VelocityPath=2; Kuka.CurrentCDSetIndex=0; Kuka.MovementParameterFieldEnabled=True; IlfCommand=LIN
;ENDFOLD
$BWDSTART = FALSE
LDAT_ACT = LCPDAT539
FDAT_ACT = FP539
BAS(#CP_PARAMS, 2.0)
SET_CD_PARAMS (0)
LIN XP539
;ENDFOLD

;FOLD LIN P540 Vel=2 m/s CPDAT540 Tool[1]:marker Base[0] ;%{PE}
;FOLD Parameters ;%{h}
;Params IlfProvider=kukaroboter.basistech.inlineforms.movement.old; Kuka.IsGlobalPoint=False; Kuka.PointName=P540; Kuka.BlendingEnabled=False; Kuka.MoveDataName=CPDAT1; Kuka.VelocityPath=2; Kuka.CurrentCDSetIndex=0; Kuka.MovementParameterFieldEnabled=True; IlfCommand=LIN
;ENDFOLD
$BWDSTART = FALSE
LDAT_ACT = LCPDAT540
FDAT_ACT = FP540
BAS(#CP_PARAMS, 2.0)
SET_CD_PARAMS (0)
LIN XP540
;ENDFOLD

;FOLD LIN P541 Vel=2 m/s CPDAT541 Tool[1]:marker Base[0] ;%{PE}
;FOLD Parameters ;%{h}
;Params IlfProvider=kukaroboter.basistech.inlineforms.movement.old; Kuka.IsGlobalPoint=False; Kuka.PointName=P541; Kuka.BlendingEnabled=False; Kuka.MoveDataName=CPDAT1; Kuka.VelocityPath=2; Kuka.CurrentCDSetIndex=0; Kuka.MovementParameterFieldEnabled=True; IlfCommand=LIN
;ENDFOLD
$BWDSTART = FALSE
LDAT_ACT = LCPDAT541
FDAT_ACT = FP541
BAS(#CP_PARAMS, 2.0)
SET_CD_PARAMS (0)
LIN XP541
;ENDFOLD

;FOLD LIN P542 Vel=2 m/s CPDAT542 Tool[1]:marker Base[0] ;%{PE}
;FOLD Parameters ;%{h}
;Params IlfProvider=kukaroboter.basistech.inlineforms.movement.old; Kuka.IsGlobalPoint=False; Kuka.PointName=P542; Kuka.BlendingEnabled=False; Kuka.MoveDataName=CPDAT1; Kuka.VelocityPath=2; Kuka.CurrentCDSetIndex=0; Kuka.MovementParameterFieldEnabled=True; IlfCommand=LIN
;ENDFOLD
$BWDSTART = FALSE
LDAT_ACT = LCPDAT542
FDAT_ACT = FP542
BAS(#CP_PARAMS, 2.0)
SET_CD_PARAMS (0)
LIN XP542
;ENDFOLD

;FOLD LIN P543 Vel=2 m/s CPDAT543 Tool[1]:marker Base[0] ;%{PE}
;FOLD Parameters ;%{h}
;Params IlfProvider=kukaroboter.basistech.inlineforms.movement.old; Kuka.IsGlobalPoint=False; Kuka.PointName=P543; Kuka.BlendingEnabled=False; Kuka.MoveDataName=CPDAT1; Kuka.VelocityPath=2; Kuka.CurrentCDSetIndex=0; Kuka.MovementParameterFieldEnabled=True; IlfCommand=LIN
;ENDFOLD
$BWDSTART = FALSE
LDAT_ACT = LCPDAT543
FDAT_ACT = FP543
BAS(#CP_PARAMS, 2.0)
SET_CD_PARAMS (0)
LIN XP543
;ENDFOLD

;FOLD LIN P544 Vel=2 m/s CPDAT544 Tool[1]:marker Base[0] ;%{PE}
;FOLD Parameters ;%{h}
;Params IlfProvider=kukaroboter.basistech.inlineforms.movement.old; Kuka.IsGlobalPoint=False; Kuka.PointName=P544; Kuka.BlendingEnabled=False; Kuka.MoveDataName=CPDAT1; Kuka.VelocityPath=2; Kuka.CurrentCDSetIndex=0; Kuka.MovementParameterFieldEnabled=True; IlfCommand=LIN
;ENDFOLD
$BWDSTART = FALSE
LDAT_ACT = LCPDAT544
FDAT_ACT = FP544
BAS(#CP_PARAMS, 2.0)
SET_CD_PARAMS (0)
LIN XP544
;ENDFOLD

;FOLD LIN P545 Vel=2 m/s CPDAT545 Tool[1]:marker Base[0] ;%{PE}
;FOLD Parameters ;%{h}
;Params IlfProvider=kukaroboter.basistech.inlineforms.movement.old; Kuka.IsGlobalPoint=False; Kuka.PointName=P545; Kuka.BlendingEnabled=False; Kuka.MoveDataName=CPDAT1; Kuka.VelocityPath=2; Kuka.CurrentCDSetIndex=0; Kuka.MovementParameterFieldEnabled=True; IlfCommand=LIN
;ENDFOLD
$BWDSTART = FALSE
LDAT_ACT = LCPDAT545
FDAT_ACT = FP545
BAS(#CP_PARAMS, 2.0)
SET_CD_PARAMS (0)
LIN XP545
;ENDFOLD

;FOLD LIN P546 Vel=2 m/s CPDAT546 Tool[1]:marker Base[0] ;%{PE}
;FOLD Parameters ;%{h}
;Params IlfProvider=kukaroboter.basistech.inlineforms.movement.old; Kuka.IsGlobalPoint=False; Kuka.PointName=P546; Kuka.BlendingEnabled=False; Kuka.MoveDataName=CPDAT1; Kuka.VelocityPath=2; Kuka.CurrentCDSetIndex=0; Kuka.MovementParameterFieldEnabled=True; IlfCommand=LIN
;ENDFOLD
$BWDSTART = FALSE
LDAT_ACT = LCPDAT546
FDAT_ACT = FP546
BAS(#CP_PARAMS, 2.0)
SET_CD_PARAMS (0)
LIN XP546
;ENDFOLD

;FOLD LIN P547 Vel=2 m/s CPDAT547 Tool[1]:marker Base[0] ;%{PE}
;FOLD Parameters ;%{h}
;Params IlfProvider=kukaroboter.basistech.inlineforms.movement.old; Kuka.IsGlobalPoint=False; Kuka.PointName=P547; Kuka.BlendingEnabled=False; Kuka.MoveDataName=CPDAT1; Kuka.VelocityPath=2; Kuka.CurrentCDSetIndex=0; Kuka.MovementParameterFieldEnabled=True; IlfCommand=LIN
;ENDFOLD
$BWDSTART = FALSE
LDAT_ACT = LCPDAT547
FDAT_ACT = FP547
BAS(#CP_PARAMS, 2.0)
SET_CD_PARAMS (0)
LIN XP547
;ENDFOLD

;FOLD LIN P548 Vel=2 m/s CPDAT548 Tool[1]:marker Base[0] ;%{PE}
;FOLD Parameters ;%{h}
;Params IlfProvider=kukaroboter.basistech.inlineforms.movement.old; Kuka.IsGlobalPoint=False; Kuka.PointName=P548; Kuka.BlendingEnabled=False; Kuka.MoveDataName=CPDAT1; Kuka.VelocityPath=2; Kuka.CurrentCDSetIndex=0; Kuka.MovementParameterFieldEnabled=True; IlfCommand=LIN
;ENDFOLD
$BWDSTART = FALSE
LDAT_ACT = LCPDAT548
FDAT_ACT = FP548
BAS(#CP_PARAMS, 2.0)
SET_CD_PARAMS (0)
LIN XP548
;ENDFOLD

;FOLD LIN P549 Vel=2 m/s CPDAT549 Tool[1]:marker Base[0] ;%{PE}
;FOLD Parameters ;%{h}
;Params IlfProvider=kukaroboter.basistech.inlineforms.movement.old; Kuka.IsGlobalPoint=False; Kuka.PointName=P549; Kuka.BlendingEnabled=False; Kuka.MoveDataName=CPDAT1; Kuka.VelocityPath=2; Kuka.CurrentCDSetIndex=0; Kuka.MovementParameterFieldEnabled=True; IlfCommand=LIN
;ENDFOLD
$BWDSTART = FALSE
LDAT_ACT = LCPDAT549
FDAT_ACT = FP549
BAS(#CP_PARAMS, 2.0)
SET_CD_PARAMS (0)
LIN XP549
;ENDFOLD

;FOLD LIN P550 Vel=2 m/s CPDAT550 Tool[1]:marker Base[0] ;%{PE}
;FOLD Parameters ;%{h}
;Params IlfProvider=kukaroboter.basistech.inlineforms.movement.old; Kuka.IsGlobalPoint=False; Kuka.PointName=P550; Kuka.BlendingEnabled=False; Kuka.MoveDataName=CPDAT1; Kuka.VelocityPath=2; Kuka.CurrentCDSetIndex=0; Kuka.MovementParameterFieldEnabled=True; IlfCommand=LIN
;ENDFOLD
$BWDSTART = FALSE
LDAT_ACT = LCPDAT550
FDAT_ACT = FP550
BAS(#CP_PARAMS, 2.0)
SET_CD_PARAMS (0)
LIN XP550
;ENDFOLD

;FOLD LIN P551 Vel=2 m/s CPDAT551 Tool[1]:marker Base[0] ;%{PE}
;FOLD Parameters ;%{h}
;Params IlfProvider=kukaroboter.basistech.inlineforms.movement.old; Kuka.IsGlobalPoint=False; Kuka.PointName=P551; Kuka.BlendingEnabled=False; Kuka.MoveDataName=CPDAT1; Kuka.VelocityPath=2; Kuka.CurrentCDSetIndex=0; Kuka.MovementParameterFieldEnabled=True; IlfCommand=LIN
;ENDFOLD
$BWDSTART = FALSE
LDAT_ACT = LCPDAT551
FDAT_ACT = FP551
BAS(#CP_PARAMS, 2.0)
SET_CD_PARAMS (0)
LIN XP551
;ENDFOLD

;FOLD LIN P552 Vel=2 m/s CPDAT552 Tool[1]:marker Base[0] ;%{PE}
;FOLD Parameters ;%{h}
;Params IlfProvider=kukaroboter.basistech.inlineforms.movement.old; Kuka.IsGlobalPoint=False; Kuka.PointName=P552; Kuka.BlendingEnabled=False; Kuka.MoveDataName=CPDAT1; Kuka.VelocityPath=2; Kuka.CurrentCDSetIndex=0; Kuka.MovementParameterFieldEnabled=True; IlfCommand=LIN
;ENDFOLD
$BWDSTART = FALSE
LDAT_ACT = LCPDAT552
FDAT_ACT = FP552
BAS(#CP_PARAMS, 2.0)
SET_CD_PARAMS (0)
LIN XP552
;ENDFOLD

;FOLD LIN P553 Vel=2 m/s CPDAT553 Tool[1]:marker Base[0] ;%{PE}
;FOLD Parameters ;%{h}
;Params IlfProvider=kukaroboter.basistech.inlineforms.movement.old; Kuka.IsGlobalPoint=False; Kuka.PointName=P553; Kuka.BlendingEnabled=False; Kuka.MoveDataName=CPDAT1; Kuka.VelocityPath=2; Kuka.CurrentCDSetIndex=0; Kuka.MovementParameterFieldEnabled=True; IlfCommand=LIN
;ENDFOLD
$BWDSTART = FALSE
LDAT_ACT = LCPDAT553
FDAT_ACT = FP553
BAS(#CP_PARAMS, 2.0)
SET_CD_PARAMS (0)
LIN XP553
;ENDFOLD

;FOLD LIN P554 Vel=2 m/s CPDAT554 Tool[1]:marker Base[0] ;%{PE}
;FOLD Parameters ;%{h}
;Params IlfProvider=kukaroboter.basistech.inlineforms.movement.old; Kuka.IsGlobalPoint=False; Kuka.PointName=P554; Kuka.BlendingEnabled=False; Kuka.MoveDataName=CPDAT1; Kuka.VelocityPath=2; Kuka.CurrentCDSetIndex=0; Kuka.MovementParameterFieldEnabled=True; IlfCommand=LIN
;ENDFOLD
$BWDSTART = FALSE
LDAT_ACT = LCPDAT554
FDAT_ACT = FP554
BAS(#CP_PARAMS, 2.0)
SET_CD_PARAMS (0)
LIN XP554
;ENDFOLD

;FOLD LIN P555 Vel=2 m/s CPDAT555 Tool[1]:marker Base[0] ;%{PE}
;FOLD Parameters ;%{h}
;Params IlfProvider=kukaroboter.basistech.inlineforms.movement.old; Kuka.IsGlobalPoint=False; Kuka.PointName=P555; Kuka.BlendingEnabled=False; Kuka.MoveDataName=CPDAT1; Kuka.VelocityPath=2; Kuka.CurrentCDSetIndex=0; Kuka.MovementParameterFieldEnabled=True; IlfCommand=LIN
;ENDFOLD
$BWDSTART = FALSE
LDAT_ACT = LCPDAT555
FDAT_ACT = FP555
BAS(#CP_PARAMS, 2.0)
SET_CD_PARAMS (0)
LIN XP555
;ENDFOLD

;FOLD LIN P556 Vel=2 m/s CPDAT556 Tool[1]:marker Base[0] ;%{PE}
;FOLD Parameters ;%{h}
;Params IlfProvider=kukaroboter.basistech.inlineforms.movement.old; Kuka.IsGlobalPoint=False; Kuka.PointName=P556; Kuka.BlendingEnabled=False; Kuka.MoveDataName=CPDAT1; Kuka.VelocityPath=2; Kuka.CurrentCDSetIndex=0; Kuka.MovementParameterFieldEnabled=True; IlfCommand=LIN
;ENDFOLD
$BWDSTART = FALSE
LDAT_ACT = LCPDAT556
FDAT_ACT = FP556
BAS(#CP_PARAMS, 2.0)
SET_CD_PARAMS (0)
LIN XP556
;ENDFOLD

;FOLD LIN P557 Vel=2 m/s CPDAT557 Tool[1]:marker Base[0] ;%{PE}
;FOLD Parameters ;%{h}
;Params IlfProvider=kukaroboter.basistech.inlineforms.movement.old; Kuka.IsGlobalPoint=False; Kuka.PointName=P557; Kuka.BlendingEnabled=False; Kuka.MoveDataName=CPDAT1; Kuka.VelocityPath=2; Kuka.CurrentCDSetIndex=0; Kuka.MovementParameterFieldEnabled=True; IlfCommand=LIN
;ENDFOLD
$BWDSTART = FALSE
LDAT_ACT = LCPDAT557
FDAT_ACT = FP557
BAS(#CP_PARAMS, 2.0)
SET_CD_PARAMS (0)
LIN XP557
;ENDFOLD

;FOLD LIN P558 Vel=2 m/s CPDAT558 Tool[1]:marker Base[0] ;%{PE}
;FOLD Parameters ;%{h}
;Params IlfProvider=kukaroboter.basistech.inlineforms.movement.old; Kuka.IsGlobalPoint=False; Kuka.PointName=P558; Kuka.BlendingEnabled=False; Kuka.MoveDataName=CPDAT1; Kuka.VelocityPath=2; Kuka.CurrentCDSetIndex=0; Kuka.MovementParameterFieldEnabled=True; IlfCommand=LIN
;ENDFOLD
$BWDSTART = FALSE
LDAT_ACT = LCPDAT558
FDAT_ACT = FP558
BAS(#CP_PARAMS, 2.0)
SET_CD_PARAMS (0)
LIN XP558
;ENDFOLD

;FOLD LIN P559 Vel=2 m/s CPDAT559 Tool[1]:marker Base[0] ;%{PE}
;FOLD Parameters ;%{h}
;Params IlfProvider=kukaroboter.basistech.inlineforms.movement.old; Kuka.IsGlobalPoint=False; Kuka.PointName=P559; Kuka.BlendingEnabled=False; Kuka.MoveDataName=CPDAT1; Kuka.VelocityPath=2; Kuka.CurrentCDSetIndex=0; Kuka.MovementParameterFieldEnabled=True; IlfCommand=LIN
;ENDFOLD
$BWDSTART = FALSE
LDAT_ACT = LCPDAT559
FDAT_ACT = FP559
BAS(#CP_PARAMS, 2.0)
SET_CD_PARAMS (0)
LIN XP559
;ENDFOLD

;FOLD LIN P560 Vel=2 m/s CPDAT560 Tool[1]:marker Base[0] ;%{PE}
;FOLD Parameters ;%{h}
;Params IlfProvider=kukaroboter.basistech.inlineforms.movement.old; Kuka.IsGlobalPoint=False; Kuka.PointName=P560; Kuka.BlendingEnabled=False; Kuka.MoveDataName=CPDAT1; Kuka.VelocityPath=2; Kuka.CurrentCDSetIndex=0; Kuka.MovementParameterFieldEnabled=True; IlfCommand=LIN
;ENDFOLD
$BWDSTART = FALSE
LDAT_ACT = LCPDAT560
FDAT_ACT = FP560
BAS(#CP_PARAMS, 2.0)
SET_CD_PARAMS (0)
LIN XP560
;ENDFOLD

;FOLD LIN P561 Vel=2 m/s CPDAT561 Tool[1]:marker Base[0] ;%{PE}
;FOLD Parameters ;%{h}
;Params IlfProvider=kukaroboter.basistech.inlineforms.movement.old; Kuka.IsGlobalPoint=False; Kuka.PointName=P561; Kuka.BlendingEnabled=False; Kuka.MoveDataName=CPDAT1; Kuka.VelocityPath=2; Kuka.CurrentCDSetIndex=0; Kuka.MovementParameterFieldEnabled=True; IlfCommand=LIN
;ENDFOLD
$BWDSTART = FALSE
LDAT_ACT = LCPDAT561
FDAT_ACT = FP561
BAS(#CP_PARAMS, 2.0)
SET_CD_PARAMS (0)
LIN XP561
;ENDFOLD

;FOLD LIN P562 Vel=2 m/s CPDAT562 Tool[1]:marker Base[0] ;%{PE}
;FOLD Parameters ;%{h}
;Params IlfProvider=kukaroboter.basistech.inlineforms.movement.old; Kuka.IsGlobalPoint=False; Kuka.PointName=P562; Kuka.BlendingEnabled=False; Kuka.MoveDataName=CPDAT1; Kuka.VelocityPath=2; Kuka.CurrentCDSetIndex=0; Kuka.MovementParameterFieldEnabled=True; IlfCommand=LIN
;ENDFOLD
$BWDSTART = FALSE
LDAT_ACT = LCPDAT562
FDAT_ACT = FP562
BAS(#CP_PARAMS, 2.0)
SET_CD_PARAMS (0)
LIN XP562
;ENDFOLD

;FOLD LIN P563 Vel=2 m/s CPDAT563 Tool[1]:marker Base[0] ;%{PE}
;FOLD Parameters ;%{h}
;Params IlfProvider=kukaroboter.basistech.inlineforms.movement.old; Kuka.IsGlobalPoint=False; Kuka.PointName=P563; Kuka.BlendingEnabled=False; Kuka.MoveDataName=CPDAT1; Kuka.VelocityPath=2; Kuka.CurrentCDSetIndex=0; Kuka.MovementParameterFieldEnabled=True; IlfCommand=LIN
;ENDFOLD
$BWDSTART = FALSE
LDAT_ACT = LCPDAT563
FDAT_ACT = FP563
BAS(#CP_PARAMS, 2.0)
SET_CD_PARAMS (0)
LIN XP563
;ENDFOLD

;FOLD LIN P564 Vel=2 m/s CPDAT564 Tool[1]:marker Base[0] ;%{PE}
;FOLD Parameters ;%{h}
;Params IlfProvider=kukaroboter.basistech.inlineforms.movement.old; Kuka.IsGlobalPoint=False; Kuka.PointName=P564; Kuka.BlendingEnabled=False; Kuka.MoveDataName=CPDAT1; Kuka.VelocityPath=2; Kuka.CurrentCDSetIndex=0; Kuka.MovementParameterFieldEnabled=True; IlfCommand=LIN
;ENDFOLD
$BWDSTART = FALSE
LDAT_ACT = LCPDAT564
FDAT_ACT = FP564
BAS(#CP_PARAMS, 2.0)
SET_CD_PARAMS (0)
LIN XP564
;ENDFOLD

;FOLD LIN P565 Vel=2 m/s CPDAT565 Tool[1]:marker Base[0] ;%{PE}
;FOLD Parameters ;%{h}
;Params IlfProvider=kukaroboter.basistech.inlineforms.movement.old; Kuka.IsGlobalPoint=False; Kuka.PointName=P565; Kuka.BlendingEnabled=False; Kuka.MoveDataName=CPDAT1; Kuka.VelocityPath=2; Kuka.CurrentCDSetIndex=0; Kuka.MovementParameterFieldEnabled=True; IlfCommand=LIN
;ENDFOLD
$BWDSTART = FALSE
LDAT_ACT = LCPDAT565
FDAT_ACT = FP565
BAS(#CP_PARAMS, 2.0)
SET_CD_PARAMS (0)
LIN XP565
;ENDFOLD

;FOLD LIN P566 Vel=2 m/s CPDAT566 Tool[1]:marker Base[0] ;%{PE}
;FOLD Parameters ;%{h}
;Params IlfProvider=kukaroboter.basistech.inlineforms.movement.old; Kuka.IsGlobalPoint=False; Kuka.PointName=P566; Kuka.BlendingEnabled=False; Kuka.MoveDataName=CPDAT1; Kuka.VelocityPath=2; Kuka.CurrentCDSetIndex=0; Kuka.MovementParameterFieldEnabled=True; IlfCommand=LIN
;ENDFOLD
$BWDSTART = FALSE
LDAT_ACT = LCPDAT566
FDAT_ACT = FP566
BAS(#CP_PARAMS, 2.0)
SET_CD_PARAMS (0)
LIN XP566
;ENDFOLD

;FOLD LIN P567 Vel=2 m/s CPDAT567 Tool[1]:marker Base[0] ;%{PE}
;FOLD Parameters ;%{h}
;Params IlfProvider=kukaroboter.basistech.inlineforms.movement.old; Kuka.IsGlobalPoint=False; Kuka.PointName=P567; Kuka.BlendingEnabled=False; Kuka.MoveDataName=CPDAT1; Kuka.VelocityPath=2; Kuka.CurrentCDSetIndex=0; Kuka.MovementParameterFieldEnabled=True; IlfCommand=LIN
;ENDFOLD
$BWDSTART = FALSE
LDAT_ACT = LCPDAT567
FDAT_ACT = FP567
BAS(#CP_PARAMS, 2.0)
SET_CD_PARAMS (0)
LIN XP567
;ENDFOLD

;FOLD LIN P568 Vel=2 m/s CPDAT568 Tool[1]:marker Base[0] ;%{PE}
;FOLD Parameters ;%{h}
;Params IlfProvider=kukaroboter.basistech.inlineforms.movement.old; Kuka.IsGlobalPoint=False; Kuka.PointName=P568; Kuka.BlendingEnabled=False; Kuka.MoveDataName=CPDAT1; Kuka.VelocityPath=2; Kuka.CurrentCDSetIndex=0; Kuka.MovementParameterFieldEnabled=True; IlfCommand=LIN
;ENDFOLD
$BWDSTART = FALSE
LDAT_ACT = LCPDAT568
FDAT_ACT = FP568
BAS(#CP_PARAMS, 2.0)
SET_CD_PARAMS (0)
LIN XP568
;ENDFOLD

;FOLD LIN P569 Vel=2 m/s CPDAT569 Tool[1]:marker Base[0] ;%{PE}
;FOLD Parameters ;%{h}
;Params IlfProvider=kukaroboter.basistech.inlineforms.movement.old; Kuka.IsGlobalPoint=False; Kuka.PointName=P569; Kuka.BlendingEnabled=False; Kuka.MoveDataName=CPDAT1; Kuka.VelocityPath=2; Kuka.CurrentCDSetIndex=0; Kuka.MovementParameterFieldEnabled=True; IlfCommand=LIN
;ENDFOLD
$BWDSTART = FALSE
LDAT_ACT = LCPDAT569
FDAT_ACT = FP569
BAS(#CP_PARAMS, 2.0)
SET_CD_PARAMS (0)
LIN XP569
;ENDFOLD

;FOLD LIN P570 Vel=2 m/s CPDAT570 Tool[1]:marker Base[0] ;%{PE}
;FOLD Parameters ;%{h}
;Params IlfProvider=kukaroboter.basistech.inlineforms.movement.old; Kuka.IsGlobalPoint=False; Kuka.PointName=P570; Kuka.BlendingEnabled=False; Kuka.MoveDataName=CPDAT1; Kuka.VelocityPath=2; Kuka.CurrentCDSetIndex=0; Kuka.MovementParameterFieldEnabled=True; IlfCommand=LIN
;ENDFOLD
$BWDSTART = FALSE
LDAT_ACT = LCPDAT570
FDAT_ACT = FP570
BAS(#CP_PARAMS, 2.0)
SET_CD_PARAMS (0)
LIN XP570
;ENDFOLD

;FOLD LIN P571 Vel=2 m/s CPDAT571 Tool[1]:marker Base[0] ;%{PE}
;FOLD Parameters ;%{h}
;Params IlfProvider=kukaroboter.basistech.inlineforms.movement.old; Kuka.IsGlobalPoint=False; Kuka.PointName=P571; Kuka.BlendingEnabled=False; Kuka.MoveDataName=CPDAT1; Kuka.VelocityPath=2; Kuka.CurrentCDSetIndex=0; Kuka.MovementParameterFieldEnabled=True; IlfCommand=LIN
;ENDFOLD
$BWDSTART = FALSE
LDAT_ACT = LCPDAT571
FDAT_ACT = FP571
BAS(#CP_PARAMS, 2.0)
SET_CD_PARAMS (0)
LIN XP571
;ENDFOLD

;FOLD LIN P572 Vel=2 m/s CPDAT572 Tool[1]:marker Base[0] ;%{PE}
;FOLD Parameters ;%{h}
;Params IlfProvider=kukaroboter.basistech.inlineforms.movement.old; Kuka.IsGlobalPoint=False; Kuka.PointName=P572; Kuka.BlendingEnabled=False; Kuka.MoveDataName=CPDAT1; Kuka.VelocityPath=2; Kuka.CurrentCDSetIndex=0; Kuka.MovementParameterFieldEnabled=True; IlfCommand=LIN
;ENDFOLD
$BWDSTART = FALSE
LDAT_ACT = LCPDAT572
FDAT_ACT = FP572
BAS(#CP_PARAMS, 2.0)
SET_CD_PARAMS (0)
LIN XP572
;ENDFOLD

;FOLD LIN P573 Vel=2 m/s CPDAT573 Tool[1]:marker Base[0] ;%{PE}
;FOLD Parameters ;%{h}
;Params IlfProvider=kukaroboter.basistech.inlineforms.movement.old; Kuka.IsGlobalPoint=False; Kuka.PointName=P573; Kuka.BlendingEnabled=False; Kuka.MoveDataName=CPDAT1; Kuka.VelocityPath=2; Kuka.CurrentCDSetIndex=0; Kuka.MovementParameterFieldEnabled=True; IlfCommand=LIN
;ENDFOLD
$BWDSTART = FALSE
LDAT_ACT = LCPDAT573
FDAT_ACT = FP573
BAS(#CP_PARAMS, 2.0)
SET_CD_PARAMS (0)
LIN XP573
;ENDFOLD

;FOLD LIN P574 Vel=2 m/s CPDAT574 Tool[1]:marker Base[0] ;%{PE}
;FOLD Parameters ;%{h}
;Params IlfProvider=kukaroboter.basistech.inlineforms.movement.old; Kuka.IsGlobalPoint=False; Kuka.PointName=P574; Kuka.BlendingEnabled=False; Kuka.MoveDataName=CPDAT1; Kuka.VelocityPath=2; Kuka.CurrentCDSetIndex=0; Kuka.MovementParameterFieldEnabled=True; IlfCommand=LIN
;ENDFOLD
$BWDSTART = FALSE
LDAT_ACT = LCPDAT574
FDAT_ACT = FP574
BAS(#CP_PARAMS, 2.0)
SET_CD_PARAMS (0)
LIN XP574
;ENDFOLD

;FOLD LIN P575 Vel=2 m/s CPDAT575 Tool[1]:marker Base[0] ;%{PE}
;FOLD Parameters ;%{h}
;Params IlfProvider=kukaroboter.basistech.inlineforms.movement.old; Kuka.IsGlobalPoint=False; Kuka.PointName=P575; Kuka.BlendingEnabled=False; Kuka.MoveDataName=CPDAT1; Kuka.VelocityPath=2; Kuka.CurrentCDSetIndex=0; Kuka.MovementParameterFieldEnabled=True; IlfCommand=LIN
;ENDFOLD
$BWDSTART = FALSE
LDAT_ACT = LCPDAT575
FDAT_ACT = FP575
BAS(#CP_PARAMS, 2.0)
SET_CD_PARAMS (0)
LIN XP575
;ENDFOLD

;FOLD LIN P576 Vel=2 m/s CPDAT576 Tool[1]:marker Base[0] ;%{PE}
;FOLD Parameters ;%{h}
;Params IlfProvider=kukaroboter.basistech.inlineforms.movement.old; Kuka.IsGlobalPoint=False; Kuka.PointName=P576; Kuka.BlendingEnabled=False; Kuka.MoveDataName=CPDAT1; Kuka.VelocityPath=2; Kuka.CurrentCDSetIndex=0; Kuka.MovementParameterFieldEnabled=True; IlfCommand=LIN
;ENDFOLD
$BWDSTART = FALSE
LDAT_ACT = LCPDAT576
FDAT_ACT = FP576
BAS(#CP_PARAMS, 2.0)
SET_CD_PARAMS (0)
LIN XP576
;ENDFOLD

;FOLD LIN P577 Vel=2 m/s CPDAT577 Tool[1]:marker Base[0] ;%{PE}
;FOLD Parameters ;%{h}
;Params IlfProvider=kukaroboter.basistech.inlineforms.movement.old; Kuka.IsGlobalPoint=False; Kuka.PointName=P577; Kuka.BlendingEnabled=False; Kuka.MoveDataName=CPDAT1; Kuka.VelocityPath=2; Kuka.CurrentCDSetIndex=0; Kuka.MovementParameterFieldEnabled=True; IlfCommand=LIN
;ENDFOLD
$BWDSTART = FALSE
LDAT_ACT = LCPDAT577
FDAT_ACT = FP577
BAS(#CP_PARAMS, 2.0)
SET_CD_PARAMS (0)
LIN XP577
;ENDFOLD

;FOLD LIN P578 Vel=2 m/s CPDAT578 Tool[1]:marker Base[0] ;%{PE}
;FOLD Parameters ;%{h}
;Params IlfProvider=kukaroboter.basistech.inlineforms.movement.old; Kuka.IsGlobalPoint=False; Kuka.PointName=P578; Kuka.BlendingEnabled=False; Kuka.MoveDataName=CPDAT1; Kuka.VelocityPath=2; Kuka.CurrentCDSetIndex=0; Kuka.MovementParameterFieldEnabled=True; IlfCommand=LIN
;ENDFOLD
$BWDSTART = FALSE
LDAT_ACT = LCPDAT578
FDAT_ACT = FP578
BAS(#CP_PARAMS, 2.0)
SET_CD_PARAMS (0)
LIN XP578
;ENDFOLD

;FOLD LIN P579 Vel=2 m/s CPDAT579 Tool[1]:marker Base[0] ;%{PE}
;FOLD Parameters ;%{h}
;Params IlfProvider=kukaroboter.basistech.inlineforms.movement.old; Kuka.IsGlobalPoint=False; Kuka.PointName=P579; Kuka.BlendingEnabled=False; Kuka.MoveDataName=CPDAT1; Kuka.VelocityPath=2; Kuka.CurrentCDSetIndex=0; Kuka.MovementParameterFieldEnabled=True; IlfCommand=LIN
;ENDFOLD
$BWDSTART = FALSE
LDAT_ACT = LCPDAT579
FDAT_ACT = FP579
BAS(#CP_PARAMS, 2.0)
SET_CD_PARAMS (0)
LIN XP579
;ENDFOLD

;FOLD LIN P580 Vel=2 m/s CPDAT580 Tool[1]:marker Base[0] ;%{PE}
;FOLD Parameters ;%{h}
;Params IlfProvider=kukaroboter.basistech.inlineforms.movement.old; Kuka.IsGlobalPoint=False; Kuka.PointName=P580; Kuka.BlendingEnabled=False; Kuka.MoveDataName=CPDAT1; Kuka.VelocityPath=2; Kuka.CurrentCDSetIndex=0; Kuka.MovementParameterFieldEnabled=True; IlfCommand=LIN
;ENDFOLD
$BWDSTART = FALSE
LDAT_ACT = LCPDAT580
FDAT_ACT = FP580
BAS(#CP_PARAMS, 2.0)
SET_CD_PARAMS (0)
LIN XP580
;ENDFOLD

;FOLD LIN P581 Vel=2 m/s CPDAT581 Tool[1]:marker Base[0] ;%{PE}
;FOLD Parameters ;%{h}
;Params IlfProvider=kukaroboter.basistech.inlineforms.movement.old; Kuka.IsGlobalPoint=False; Kuka.PointName=P581; Kuka.BlendingEnabled=False; Kuka.MoveDataName=CPDAT1; Kuka.VelocityPath=2; Kuka.CurrentCDSetIndex=0; Kuka.MovementParameterFieldEnabled=True; IlfCommand=LIN
;ENDFOLD
$BWDSTART = FALSE
LDAT_ACT = LCPDAT581
FDAT_ACT = FP581
BAS(#CP_PARAMS, 2.0)
SET_CD_PARAMS (0)
LIN XP581
;ENDFOLD

;FOLD LIN P582 Vel=2 m/s CPDAT582 Tool[1]:marker Base[0] ;%{PE}
;FOLD Parameters ;%{h}
;Params IlfProvider=kukaroboter.basistech.inlineforms.movement.old; Kuka.IsGlobalPoint=False; Kuka.PointName=P582; Kuka.BlendingEnabled=False; Kuka.MoveDataName=CPDAT1; Kuka.VelocityPath=2; Kuka.CurrentCDSetIndex=0; Kuka.MovementParameterFieldEnabled=True; IlfCommand=LIN
;ENDFOLD
$BWDSTART = FALSE
LDAT_ACT = LCPDAT582
FDAT_ACT = FP582
BAS(#CP_PARAMS, 2.0)
SET_CD_PARAMS (0)
LIN XP582
;ENDFOLD

;FOLD LIN P583 Vel=2 m/s CPDAT583 Tool[1]:marker Base[0] ;%{PE}
;FOLD Parameters ;%{h}
;Params IlfProvider=kukaroboter.basistech.inlineforms.movement.old; Kuka.IsGlobalPoint=False; Kuka.PointName=P583; Kuka.BlendingEnabled=False; Kuka.MoveDataName=CPDAT1; Kuka.VelocityPath=2; Kuka.CurrentCDSetIndex=0; Kuka.MovementParameterFieldEnabled=True; IlfCommand=LIN
;ENDFOLD
$BWDSTART = FALSE
LDAT_ACT = LCPDAT583
FDAT_ACT = FP583
BAS(#CP_PARAMS, 2.0)
SET_CD_PARAMS (0)
LIN XP583
;ENDFOLD

;FOLD LIN P584 Vel=2 m/s CPDAT584 Tool[1]:marker Base[0] ;%{PE}
;FOLD Parameters ;%{h}
;Params IlfProvider=kukaroboter.basistech.inlineforms.movement.old; Kuka.IsGlobalPoint=False; Kuka.PointName=P584; Kuka.BlendingEnabled=False; Kuka.MoveDataName=CPDAT1; Kuka.VelocityPath=2; Kuka.CurrentCDSetIndex=0; Kuka.MovementParameterFieldEnabled=True; IlfCommand=LIN
;ENDFOLD
$BWDSTART = FALSE
LDAT_ACT = LCPDAT584
FDAT_ACT = FP584
BAS(#CP_PARAMS, 2.0)
SET_CD_PARAMS (0)
LIN XP584
;ENDFOLD

;FOLD LIN P585 Vel=2 m/s CPDAT585 Tool[1]:marker Base[0] ;%{PE}
;FOLD Parameters ;%{h}
;Params IlfProvider=kukaroboter.basistech.inlineforms.movement.old; Kuka.IsGlobalPoint=False; Kuka.PointName=P585; Kuka.BlendingEnabled=False; Kuka.MoveDataName=CPDAT1; Kuka.VelocityPath=2; Kuka.CurrentCDSetIndex=0; Kuka.MovementParameterFieldEnabled=True; IlfCommand=LIN
;ENDFOLD
$BWDSTART = FALSE
LDAT_ACT = LCPDAT585
FDAT_ACT = FP585
BAS(#CP_PARAMS, 2.0)
SET_CD_PARAMS (0)
LIN XP585
;ENDFOLD

;FOLD LIN P586 Vel=2 m/s CPDAT586 Tool[1]:marker Base[0] ;%{PE}
;FOLD Parameters ;%{h}
;Params IlfProvider=kukaroboter.basistech.inlineforms.movement.old; Kuka.IsGlobalPoint=False; Kuka.PointName=P586; Kuka.BlendingEnabled=False; Kuka.MoveDataName=CPDAT1; Kuka.VelocityPath=2; Kuka.CurrentCDSetIndex=0; Kuka.MovementParameterFieldEnabled=True; IlfCommand=LIN
;ENDFOLD
$BWDSTART = FALSE
LDAT_ACT = LCPDAT586
FDAT_ACT = FP586
BAS(#CP_PARAMS, 2.0)
SET_CD_PARAMS (0)
LIN XP586
;ENDFOLD

;FOLD LIN P587 Vel=2 m/s CPDAT587 Tool[1]:marker Base[0] ;%{PE}
;FOLD Parameters ;%{h}
;Params IlfProvider=kukaroboter.basistech.inlineforms.movement.old; Kuka.IsGlobalPoint=False; Kuka.PointName=P587; Kuka.BlendingEnabled=False; Kuka.MoveDataName=CPDAT1; Kuka.VelocityPath=2; Kuka.CurrentCDSetIndex=0; Kuka.MovementParameterFieldEnabled=True; IlfCommand=LIN
;ENDFOLD
$BWDSTART = FALSE
LDAT_ACT = LCPDAT587
FDAT_ACT = FP587
BAS(#CP_PARAMS, 2.0)
SET_CD_PARAMS (0)
LIN XP587
;ENDFOLD

;FOLD LIN P588 Vel=2 m/s CPDAT588 Tool[1]:marker Base[0] ;%{PE}
;FOLD Parameters ;%{h}
;Params IlfProvider=kukaroboter.basistech.inlineforms.movement.old; Kuka.IsGlobalPoint=False; Kuka.PointName=P588; Kuka.BlendingEnabled=False; Kuka.MoveDataName=CPDAT1; Kuka.VelocityPath=2; Kuka.CurrentCDSetIndex=0; Kuka.MovementParameterFieldEnabled=True; IlfCommand=LIN
;ENDFOLD
$BWDSTART = FALSE
LDAT_ACT = LCPDAT588
FDAT_ACT = FP588
BAS(#CP_PARAMS, 2.0)
SET_CD_PARAMS (0)
LIN XP588
;ENDFOLD

;FOLD LIN P589 Vel=2 m/s CPDAT589 Tool[1]:marker Base[0] ;%{PE}
;FOLD Parameters ;%{h}
;Params IlfProvider=kukaroboter.basistech.inlineforms.movement.old; Kuka.IsGlobalPoint=False; Kuka.PointName=P589; Kuka.BlendingEnabled=False; Kuka.MoveDataName=CPDAT1; Kuka.VelocityPath=2; Kuka.CurrentCDSetIndex=0; Kuka.MovementParameterFieldEnabled=True; IlfCommand=LIN
;ENDFOLD
$BWDSTART = FALSE
LDAT_ACT = LCPDAT589
FDAT_ACT = FP589
BAS(#CP_PARAMS, 2.0)
SET_CD_PARAMS (0)
LIN XP589
;ENDFOLD

;FOLD LIN P590 Vel=2 m/s CPDAT590 Tool[1]:marker Base[0] ;%{PE}
;FOLD Parameters ;%{h}
;Params IlfProvider=kukaroboter.basistech.inlineforms.movement.old; Kuka.IsGlobalPoint=False; Kuka.PointName=P590; Kuka.BlendingEnabled=False; Kuka.MoveDataName=CPDAT1; Kuka.VelocityPath=2; Kuka.CurrentCDSetIndex=0; Kuka.MovementParameterFieldEnabled=True; IlfCommand=LIN
;ENDFOLD
$BWDSTART = FALSE
LDAT_ACT = LCPDAT590
FDAT_ACT = FP590
BAS(#CP_PARAMS, 2.0)
SET_CD_PARAMS (0)
LIN XP590
;ENDFOLD

;FOLD LIN P591 Vel=2 m/s CPDAT591 Tool[1]:marker Base[0] ;%{PE}
;FOLD Parameters ;%{h}
;Params IlfProvider=kukaroboter.basistech.inlineforms.movement.old; Kuka.IsGlobalPoint=False; Kuka.PointName=P591; Kuka.BlendingEnabled=False; Kuka.MoveDataName=CPDAT1; Kuka.VelocityPath=2; Kuka.CurrentCDSetIndex=0; Kuka.MovementParameterFieldEnabled=True; IlfCommand=LIN
;ENDFOLD
$BWDSTART = FALSE
LDAT_ACT = LCPDAT591
FDAT_ACT = FP591
BAS(#CP_PARAMS, 2.0)
SET_CD_PARAMS (0)
LIN XP591
;ENDFOLD

;FOLD LIN P592 Vel=2 m/s CPDAT592 Tool[1]:marker Base[0] ;%{PE}
;FOLD Parameters ;%{h}
;Params IlfProvider=kukaroboter.basistech.inlineforms.movement.old; Kuka.IsGlobalPoint=False; Kuka.PointName=P592; Kuka.BlendingEnabled=False; Kuka.MoveDataName=CPDAT1; Kuka.VelocityPath=2; Kuka.CurrentCDSetIndex=0; Kuka.MovementParameterFieldEnabled=True; IlfCommand=LIN
;ENDFOLD
$BWDSTART = FALSE
LDAT_ACT = LCPDAT592
FDAT_ACT = FP592
BAS(#CP_PARAMS, 2.0)
SET_CD_PARAMS (0)
LIN XP592
;ENDFOLD

;FOLD LIN P593 Vel=2 m/s CPDAT593 Tool[1]:marker Base[0] ;%{PE}
;FOLD Parameters ;%{h}
;Params IlfProvider=kukaroboter.basistech.inlineforms.movement.old; Kuka.IsGlobalPoint=False; Kuka.PointName=P593; Kuka.BlendingEnabled=False; Kuka.MoveDataName=CPDAT1; Kuka.VelocityPath=2; Kuka.CurrentCDSetIndex=0; Kuka.MovementParameterFieldEnabled=True; IlfCommand=LIN
;ENDFOLD
$BWDSTART = FALSE
LDAT_ACT = LCPDAT593
FDAT_ACT = FP593
BAS(#CP_PARAMS, 2.0)
SET_CD_PARAMS (0)
LIN XP593
;ENDFOLD

;FOLD LIN P594 Vel=2 m/s CPDAT594 Tool[1]:marker Base[0] ;%{PE}
;FOLD Parameters ;%{h}
;Params IlfProvider=kukaroboter.basistech.inlineforms.movement.old; Kuka.IsGlobalPoint=False; Kuka.PointName=P594; Kuka.BlendingEnabled=False; Kuka.MoveDataName=CPDAT1; Kuka.VelocityPath=2; Kuka.CurrentCDSetIndex=0; Kuka.MovementParameterFieldEnabled=True; IlfCommand=LIN
;ENDFOLD
$BWDSTART = FALSE
LDAT_ACT = LCPDAT594
FDAT_ACT = FP594
BAS(#CP_PARAMS, 2.0)
SET_CD_PARAMS (0)
LIN XP594
;ENDFOLD

;FOLD LIN P595 Vel=2 m/s CPDAT595 Tool[1]:marker Base[0] ;%{PE}
;FOLD Parameters ;%{h}
;Params IlfProvider=kukaroboter.basistech.inlineforms.movement.old; Kuka.IsGlobalPoint=False; Kuka.PointName=P595; Kuka.BlendingEnabled=False; Kuka.MoveDataName=CPDAT1; Kuka.VelocityPath=2; Kuka.CurrentCDSetIndex=0; Kuka.MovementParameterFieldEnabled=True; IlfCommand=LIN
;ENDFOLD
$BWDSTART = FALSE
LDAT_ACT = LCPDAT595
FDAT_ACT = FP595
BAS(#CP_PARAMS, 2.0)
SET_CD_PARAMS (0)
LIN XP595
;ENDFOLD

;FOLD LIN P596 Vel=2 m/s CPDAT596 Tool[1]:marker Base[0] ;%{PE}
;FOLD Parameters ;%{h}
;Params IlfProvider=kukaroboter.basistech.inlineforms.movement.old; Kuka.IsGlobalPoint=False; Kuka.PointName=P596; Kuka.BlendingEnabled=False; Kuka.MoveDataName=CPDAT1; Kuka.VelocityPath=2; Kuka.CurrentCDSetIndex=0; Kuka.MovementParameterFieldEnabled=True; IlfCommand=LIN
;ENDFOLD
$BWDSTART = FALSE
LDAT_ACT = LCPDAT596
FDAT_ACT = FP596
BAS(#CP_PARAMS, 2.0)
SET_CD_PARAMS (0)
LIN XP596
;ENDFOLD

;FOLD LIN P597 Vel=2 m/s CPDAT597 Tool[1]:marker Base[0] ;%{PE}
;FOLD Parameters ;%{h}
;Params IlfProvider=kukaroboter.basistech.inlineforms.movement.old; Kuka.IsGlobalPoint=False; Kuka.PointName=P597; Kuka.BlendingEnabled=False; Kuka.MoveDataName=CPDAT1; Kuka.VelocityPath=2; Kuka.CurrentCDSetIndex=0; Kuka.MovementParameterFieldEnabled=True; IlfCommand=LIN
;ENDFOLD
$BWDSTART = FALSE
LDAT_ACT = LCPDAT597
FDAT_ACT = FP597
BAS(#CP_PARAMS, 2.0)
SET_CD_PARAMS (0)
LIN XP597
;ENDFOLD

;FOLD LIN P598 Vel=2 m/s CPDAT598 Tool[1]:marker Base[0] ;%{PE}
;FOLD Parameters ;%{h}
;Params IlfProvider=kukaroboter.basistech.inlineforms.movement.old; Kuka.IsGlobalPoint=False; Kuka.PointName=P598; Kuka.BlendingEnabled=False; Kuka.MoveDataName=CPDAT1; Kuka.VelocityPath=2; Kuka.CurrentCDSetIndex=0; Kuka.MovementParameterFieldEnabled=True; IlfCommand=LIN
;ENDFOLD
$BWDSTART = FALSE
LDAT_ACT = LCPDAT598
FDAT_ACT = FP598
BAS(#CP_PARAMS, 2.0)
SET_CD_PARAMS (0)
LIN XP598
;ENDFOLD

;FOLD LIN P599 Vel=2 m/s CPDAT599 Tool[1]:marker Base[0] ;%{PE}
;FOLD Parameters ;%{h}
;Params IlfProvider=kukaroboter.basistech.inlineforms.movement.old; Kuka.IsGlobalPoint=False; Kuka.PointName=P599; Kuka.BlendingEnabled=False; Kuka.MoveDataName=CPDAT1; Kuka.VelocityPath=2; Kuka.CurrentCDSetIndex=0; Kuka.MovementParameterFieldEnabled=True; IlfCommand=LIN
;ENDFOLD
$BWDSTART = FALSE
LDAT_ACT = LCPDAT599
FDAT_ACT = FP599
BAS(#CP_PARAMS, 2.0)
SET_CD_PARAMS (0)
LIN XP599
;ENDFOLD

;FOLD LIN P600 Vel=2 m/s CPDAT600 Tool[1]:marker Base[0] ;%{PE}
;FOLD Parameters ;%{h}
;Params IlfProvider=kukaroboter.basistech.inlineforms.movement.old; Kuka.IsGlobalPoint=False; Kuka.PointName=P600; Kuka.BlendingEnabled=False; Kuka.MoveDataName=CPDAT1; Kuka.VelocityPath=2; Kuka.CurrentCDSetIndex=0; Kuka.MovementParameterFieldEnabled=True; IlfCommand=LIN
;ENDFOLD
$BWDSTART = FALSE
LDAT_ACT = LCPDAT600
FDAT_ACT = FP600
BAS(#CP_PARAMS, 2.0)
SET_CD_PARAMS (0)
LIN XP600
;ENDFOLD

;FOLD LIN P601 Vel=2 m/s CPDAT601 Tool[1]:marker Base[0] ;%{PE}
;FOLD Parameters ;%{h}
;Params IlfProvider=kukaroboter.basistech.inlineforms.movement.old; Kuka.IsGlobalPoint=False; Kuka.PointName=P601; Kuka.BlendingEnabled=False; Kuka.MoveDataName=CPDAT1; Kuka.VelocityPath=2; Kuka.CurrentCDSetIndex=0; Kuka.MovementParameterFieldEnabled=True; IlfCommand=LIN
;ENDFOLD
$BWDSTART = FALSE
LDAT_ACT = LCPDAT601
FDAT_ACT = FP601
BAS(#CP_PARAMS, 2.0)
SET_CD_PARAMS (0)
LIN XP601
;ENDFOLD

;FOLD LIN P602 Vel=2 m/s CPDAT602 Tool[1]:marker Base[0] ;%{PE}
;FOLD Parameters ;%{h}
;Params IlfProvider=kukaroboter.basistech.inlineforms.movement.old; Kuka.IsGlobalPoint=False; Kuka.PointName=P602; Kuka.BlendingEnabled=False; Kuka.MoveDataName=CPDAT1; Kuka.VelocityPath=2; Kuka.CurrentCDSetIndex=0; Kuka.MovementParameterFieldEnabled=True; IlfCommand=LIN
;ENDFOLD
$BWDSTART = FALSE
LDAT_ACT = LCPDAT602
FDAT_ACT = FP602
BAS(#CP_PARAMS, 2.0)
SET_CD_PARAMS (0)
LIN XP602
;ENDFOLD

;FOLD LIN P603 Vel=2 m/s CPDAT603 Tool[1]:marker Base[0] ;%{PE}
;FOLD Parameters ;%{h}
;Params IlfProvider=kukaroboter.basistech.inlineforms.movement.old; Kuka.IsGlobalPoint=False; Kuka.PointName=P603; Kuka.BlendingEnabled=False; Kuka.MoveDataName=CPDAT1; Kuka.VelocityPath=2; Kuka.CurrentCDSetIndex=0; Kuka.MovementParameterFieldEnabled=True; IlfCommand=LIN
;ENDFOLD
$BWDSTART = FALSE
LDAT_ACT = LCPDAT603
FDAT_ACT = FP603
BAS(#CP_PARAMS, 2.0)
SET_CD_PARAMS (0)
LIN XP603
;ENDFOLD

;FOLD LIN P604 Vel=2 m/s CPDAT604 Tool[1]:marker Base[0] ;%{PE}
;FOLD Parameters ;%{h}
;Params IlfProvider=kukaroboter.basistech.inlineforms.movement.old; Kuka.IsGlobalPoint=False; Kuka.PointName=P604; Kuka.BlendingEnabled=False; Kuka.MoveDataName=CPDAT1; Kuka.VelocityPath=2; Kuka.CurrentCDSetIndex=0; Kuka.MovementParameterFieldEnabled=True; IlfCommand=LIN
;ENDFOLD
$BWDSTART = FALSE
LDAT_ACT = LCPDAT604
FDAT_ACT = FP604
BAS(#CP_PARAMS, 2.0)
SET_CD_PARAMS (0)
LIN XP604
;ENDFOLD

;FOLD LIN P605 Vel=2 m/s CPDAT605 Tool[1]:marker Base[0] ;%{PE}
;FOLD Parameters ;%{h}
;Params IlfProvider=kukaroboter.basistech.inlineforms.movement.old; Kuka.IsGlobalPoint=False; Kuka.PointName=P605; Kuka.BlendingEnabled=False; Kuka.MoveDataName=CPDAT1; Kuka.VelocityPath=2; Kuka.CurrentCDSetIndex=0; Kuka.MovementParameterFieldEnabled=True; IlfCommand=LIN
;ENDFOLD
$BWDSTART = FALSE
LDAT_ACT = LCPDAT605
FDAT_ACT = FP605
BAS(#CP_PARAMS, 2.0)
SET_CD_PARAMS (0)
LIN XP605
;ENDFOLD

;FOLD LIN P606 Vel=2 m/s CPDAT606 Tool[1]:marker Base[0] ;%{PE}
;FOLD Parameters ;%{h}
;Params IlfProvider=kukaroboter.basistech.inlineforms.movement.old; Kuka.IsGlobalPoint=False; Kuka.PointName=P606; Kuka.BlendingEnabled=False; Kuka.MoveDataName=CPDAT1; Kuka.VelocityPath=2; Kuka.CurrentCDSetIndex=0; Kuka.MovementParameterFieldEnabled=True; IlfCommand=LIN
;ENDFOLD
$BWDSTART = FALSE
LDAT_ACT = LCPDAT606
FDAT_ACT = FP606
BAS(#CP_PARAMS, 2.0)
SET_CD_PARAMS (0)
LIN XP606
;ENDFOLD

;FOLD LIN P607 Vel=2 m/s CPDAT607 Tool[1]:marker Base[0] ;%{PE}
;FOLD Parameters ;%{h}
;Params IlfProvider=kukaroboter.basistech.inlineforms.movement.old; Kuka.IsGlobalPoint=False; Kuka.PointName=P607; Kuka.BlendingEnabled=False; Kuka.MoveDataName=CPDAT1; Kuka.VelocityPath=2; Kuka.CurrentCDSetIndex=0; Kuka.MovementParameterFieldEnabled=True; IlfCommand=LIN
;ENDFOLD
$BWDSTART = FALSE
LDAT_ACT = LCPDAT607
FDAT_ACT = FP607
BAS(#CP_PARAMS, 2.0)
SET_CD_PARAMS (0)
LIN XP607
;ENDFOLD

;FOLD LIN P608 Vel=2 m/s CPDAT608 Tool[1]:marker Base[0] ;%{PE}
;FOLD Parameters ;%{h}
;Params IlfProvider=kukaroboter.basistech.inlineforms.movement.old; Kuka.IsGlobalPoint=False; Kuka.PointName=P608; Kuka.BlendingEnabled=False; Kuka.MoveDataName=CPDAT1; Kuka.VelocityPath=2; Kuka.CurrentCDSetIndex=0; Kuka.MovementParameterFieldEnabled=True; IlfCommand=LIN
;ENDFOLD
$BWDSTART = FALSE
LDAT_ACT = LCPDAT608
FDAT_ACT = FP608
BAS(#CP_PARAMS, 2.0)
SET_CD_PARAMS (0)
LIN XP608
;ENDFOLD

;FOLD LIN P609 Vel=2 m/s CPDAT609 Tool[1]:marker Base[0] ;%{PE}
;FOLD Parameters ;%{h}
;Params IlfProvider=kukaroboter.basistech.inlineforms.movement.old; Kuka.IsGlobalPoint=False; Kuka.PointName=P609; Kuka.BlendingEnabled=False; Kuka.MoveDataName=CPDAT1; Kuka.VelocityPath=2; Kuka.CurrentCDSetIndex=0; Kuka.MovementParameterFieldEnabled=True; IlfCommand=LIN
;ENDFOLD
$BWDSTART = FALSE
LDAT_ACT = LCPDAT609
FDAT_ACT = FP609
BAS(#CP_PARAMS, 2.0)
SET_CD_PARAMS (0)
LIN XP609
;ENDFOLD

;FOLD LIN P610 Vel=2 m/s CPDAT610 Tool[1]:marker Base[0] ;%{PE}
;FOLD Parameters ;%{h}
;Params IlfProvider=kukaroboter.basistech.inlineforms.movement.old; Kuka.IsGlobalPoint=False; Kuka.PointName=P610; Kuka.BlendingEnabled=False; Kuka.MoveDataName=CPDAT1; Kuka.VelocityPath=2; Kuka.CurrentCDSetIndex=0; Kuka.MovementParameterFieldEnabled=True; IlfCommand=LIN
;ENDFOLD
$BWDSTART = FALSE
LDAT_ACT = LCPDAT610
FDAT_ACT = FP610
BAS(#CP_PARAMS, 2.0)
SET_CD_PARAMS (0)
LIN XP610
;ENDFOLD

;FOLD LIN P611 Vel=2 m/s CPDAT611 Tool[1]:marker Base[0] ;%{PE}
;FOLD Parameters ;%{h}
;Params IlfProvider=kukaroboter.basistech.inlineforms.movement.old; Kuka.IsGlobalPoint=False; Kuka.PointName=P611; Kuka.BlendingEnabled=False; Kuka.MoveDataName=CPDAT1; Kuka.VelocityPath=2; Kuka.CurrentCDSetIndex=0; Kuka.MovementParameterFieldEnabled=True; IlfCommand=LIN
;ENDFOLD
$BWDSTART = FALSE
LDAT_ACT = LCPDAT611
FDAT_ACT = FP611
BAS(#CP_PARAMS, 2.0)
SET_CD_PARAMS (0)
LIN XP611
;ENDFOLD

;FOLD LIN P612 Vel=2 m/s CPDAT612 Tool[1]:marker Base[0] ;%{PE}
;FOLD Parameters ;%{h}
;Params IlfProvider=kukaroboter.basistech.inlineforms.movement.old; Kuka.IsGlobalPoint=False; Kuka.PointName=P612; Kuka.BlendingEnabled=False; Kuka.MoveDataName=CPDAT1; Kuka.VelocityPath=2; Kuka.CurrentCDSetIndex=0; Kuka.MovementParameterFieldEnabled=True; IlfCommand=LIN
;ENDFOLD
$BWDSTART = FALSE
LDAT_ACT = LCPDAT612
FDAT_ACT = FP612
BAS(#CP_PARAMS, 2.0)
SET_CD_PARAMS (0)
LIN XP612
;ENDFOLD

;FOLD LIN P613 Vel=2 m/s CPDAT613 Tool[1]:marker Base[0] ;%{PE}
;FOLD Parameters ;%{h}
;Params IlfProvider=kukaroboter.basistech.inlineforms.movement.old; Kuka.IsGlobalPoint=False; Kuka.PointName=P613; Kuka.BlendingEnabled=False; Kuka.MoveDataName=CPDAT1; Kuka.VelocityPath=2; Kuka.CurrentCDSetIndex=0; Kuka.MovementParameterFieldEnabled=True; IlfCommand=LIN
;ENDFOLD
$BWDSTART = FALSE
LDAT_ACT = LCPDAT613
FDAT_ACT = FP613
BAS(#CP_PARAMS, 2.0)
SET_CD_PARAMS (0)
LIN XP613
;ENDFOLD

;FOLD LIN P614 Vel=2 m/s CPDAT614 Tool[1]:marker Base[0] ;%{PE}
;FOLD Parameters ;%{h}
;Params IlfProvider=kukaroboter.basistech.inlineforms.movement.old; Kuka.IsGlobalPoint=False; Kuka.PointName=P614; Kuka.BlendingEnabled=False; Kuka.MoveDataName=CPDAT1; Kuka.VelocityPath=2; Kuka.CurrentCDSetIndex=0; Kuka.MovementParameterFieldEnabled=True; IlfCommand=LIN
;ENDFOLD
$BWDSTART = FALSE
LDAT_ACT = LCPDAT614
FDAT_ACT = FP614
BAS(#CP_PARAMS, 2.0)
SET_CD_PARAMS (0)
LIN XP614
;ENDFOLD

;FOLD LIN P615 Vel=2 m/s CPDAT615 Tool[1]:marker Base[0] ;%{PE}
;FOLD Parameters ;%{h}
;Params IlfProvider=kukaroboter.basistech.inlineforms.movement.old; Kuka.IsGlobalPoint=False; Kuka.PointName=P615; Kuka.BlendingEnabled=False; Kuka.MoveDataName=CPDAT1; Kuka.VelocityPath=2; Kuka.CurrentCDSetIndex=0; Kuka.MovementParameterFieldEnabled=True; IlfCommand=LIN
;ENDFOLD
$BWDSTART = FALSE
LDAT_ACT = LCPDAT615
FDAT_ACT = FP615
BAS(#CP_PARAMS, 2.0)
SET_CD_PARAMS (0)
LIN XP615
;ENDFOLD

;FOLD LIN P616 Vel=2 m/s CPDAT616 Tool[1]:marker Base[0] ;%{PE}
;FOLD Parameters ;%{h}
;Params IlfProvider=kukaroboter.basistech.inlineforms.movement.old; Kuka.IsGlobalPoint=False; Kuka.PointName=P616; Kuka.BlendingEnabled=False; Kuka.MoveDataName=CPDAT1; Kuka.VelocityPath=2; Kuka.CurrentCDSetIndex=0; Kuka.MovementParameterFieldEnabled=True; IlfCommand=LIN
;ENDFOLD
$BWDSTART = FALSE
LDAT_ACT = LCPDAT616
FDAT_ACT = FP616
BAS(#CP_PARAMS, 2.0)
SET_CD_PARAMS (0)
LIN XP616
;ENDFOLD

;FOLD LIN P617 Vel=2 m/s CPDAT617 Tool[1]:marker Base[0] ;%{PE}
;FOLD Parameters ;%{h}
;Params IlfProvider=kukaroboter.basistech.inlineforms.movement.old; Kuka.IsGlobalPoint=False; Kuka.PointName=P617; Kuka.BlendingEnabled=False; Kuka.MoveDataName=CPDAT1; Kuka.VelocityPath=2; Kuka.CurrentCDSetIndex=0; Kuka.MovementParameterFieldEnabled=True; IlfCommand=LIN
;ENDFOLD
$BWDSTART = FALSE
LDAT_ACT = LCPDAT617
FDAT_ACT = FP617
BAS(#CP_PARAMS, 2.0)
SET_CD_PARAMS (0)
LIN XP617
;ENDFOLD

;FOLD LIN P618 Vel=2 m/s CPDAT618 Tool[1]:marker Base[0] ;%{PE}
;FOLD Parameters ;%{h}
;Params IlfProvider=kukaroboter.basistech.inlineforms.movement.old; Kuka.IsGlobalPoint=False; Kuka.PointName=P618; Kuka.BlendingEnabled=False; Kuka.MoveDataName=CPDAT1; Kuka.VelocityPath=2; Kuka.CurrentCDSetIndex=0; Kuka.MovementParameterFieldEnabled=True; IlfCommand=LIN
;ENDFOLD
$BWDSTART = FALSE
LDAT_ACT = LCPDAT618
FDAT_ACT = FP618
BAS(#CP_PARAMS, 2.0)
SET_CD_PARAMS (0)
LIN XP618
;ENDFOLD

;FOLD LIN P619 Vel=2 m/s CPDAT619 Tool[1]:marker Base[0] ;%{PE}
;FOLD Parameters ;%{h}
;Params IlfProvider=kukaroboter.basistech.inlineforms.movement.old; Kuka.IsGlobalPoint=False; Kuka.PointName=P619; Kuka.BlendingEnabled=False; Kuka.MoveDataName=CPDAT1; Kuka.VelocityPath=2; Kuka.CurrentCDSetIndex=0; Kuka.MovementParameterFieldEnabled=True; IlfCommand=LIN
;ENDFOLD
$BWDSTART = FALSE
LDAT_ACT = LCPDAT619
FDAT_ACT = FP619
BAS(#CP_PARAMS, 2.0)
SET_CD_PARAMS (0)
LIN XP619
;ENDFOLD

